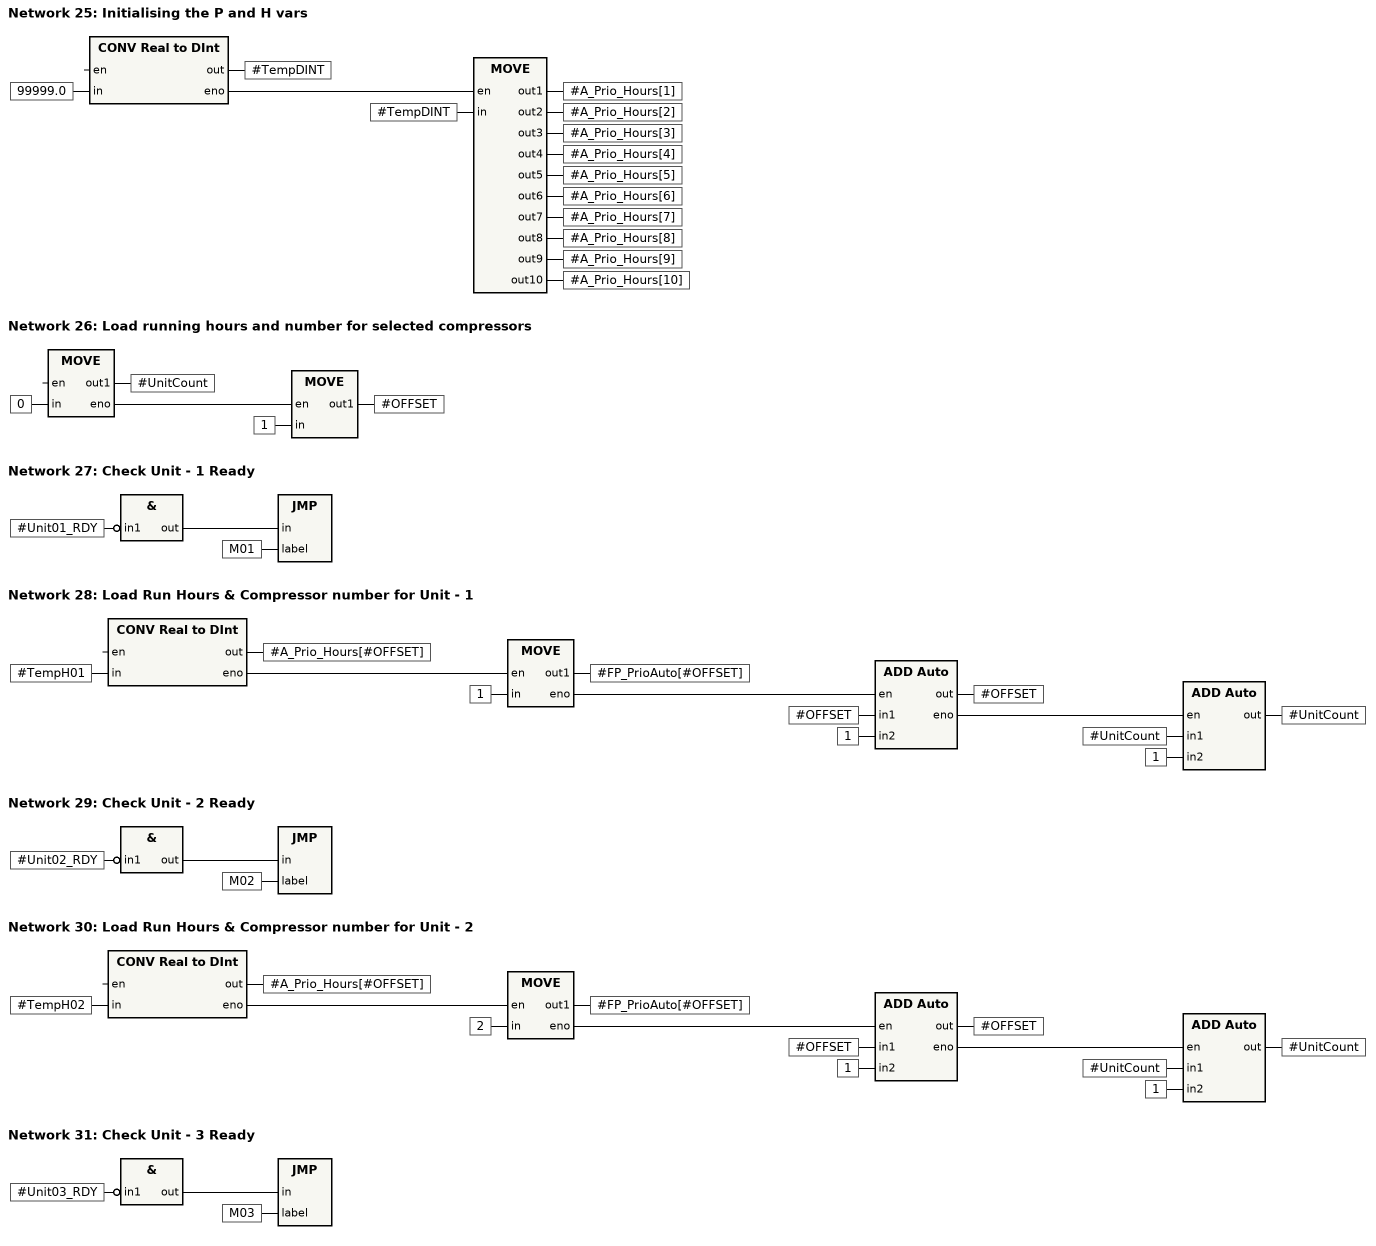
   #TempDINT := REAL_TO_DINT(99999.0);
   #A_Prio_Hours[1] := #TempDINT;
   #A_Prio_Hours[2] := #TempDINT;
   #A_Prio_Hours[3] := #TempDINT;
   #A_Prio_Hours[4] := #TempDINT;
   #A_Prio_Hours[5] := #TempDINT;
   #A_Prio_Hours[6] := #TempDINT;
   #A_Prio_Hours[7] := #TempDINT;
   #A_Prio_Hours[8] := #TempDINT;
   #A_Prio_Hours[9] := #TempDINT;
   #A_Prio_Hours[10] := #TempDINT;
END_REGION

REGION Network 26: Load running hours and number for selected compressors
   // Initialise Unit Count and Offset
   #UnitCount := 0;
   #OFFSET := 1;
END_REGION

REGION Network 27: Check Unit - 1 Ready
   IF NOT #Unit01_RDY THEN GOTO M01; END_IF;
END_REGION

REGION Network 28: Load Run Hours & Compressor number for Unit - 1
   #A_Prio_Hours[#OFFSET] := REAL_TO_DINT(#TempH01);
   #FP_PrioAuto[#OFFSET] := 1;
   #OFFSET := #OFFSET + 1;
   #UnitCount := #UnitCount + 1;
END_REGION

REGION Network 29: Check Unit - 2 Ready
   M01:
   IF NOT #Unit02_RDY THEN GOTO M02; END_IF;
END_REGION

REGION Network 30: Load Run Hours & Compressor number for Unit - 2
   #A_Prio_Hours[#OFFSET] := REAL_TO_DINT(#TempH02);
   #FP_PrioAuto[#OFFSET] := 2;
   #OFFSET := #OFFSET + 1;
   #UnitCount := #UnitCount + 1;
END_REGION

REGION Network 31: Check Unit - 3 Ready
   M02:
   IF NOT #Unit03_RDY THEN GOTO M03; END_IF;
END_REGION

REGION Network 32: Load Run Hours & Compressor number for Unit - 3
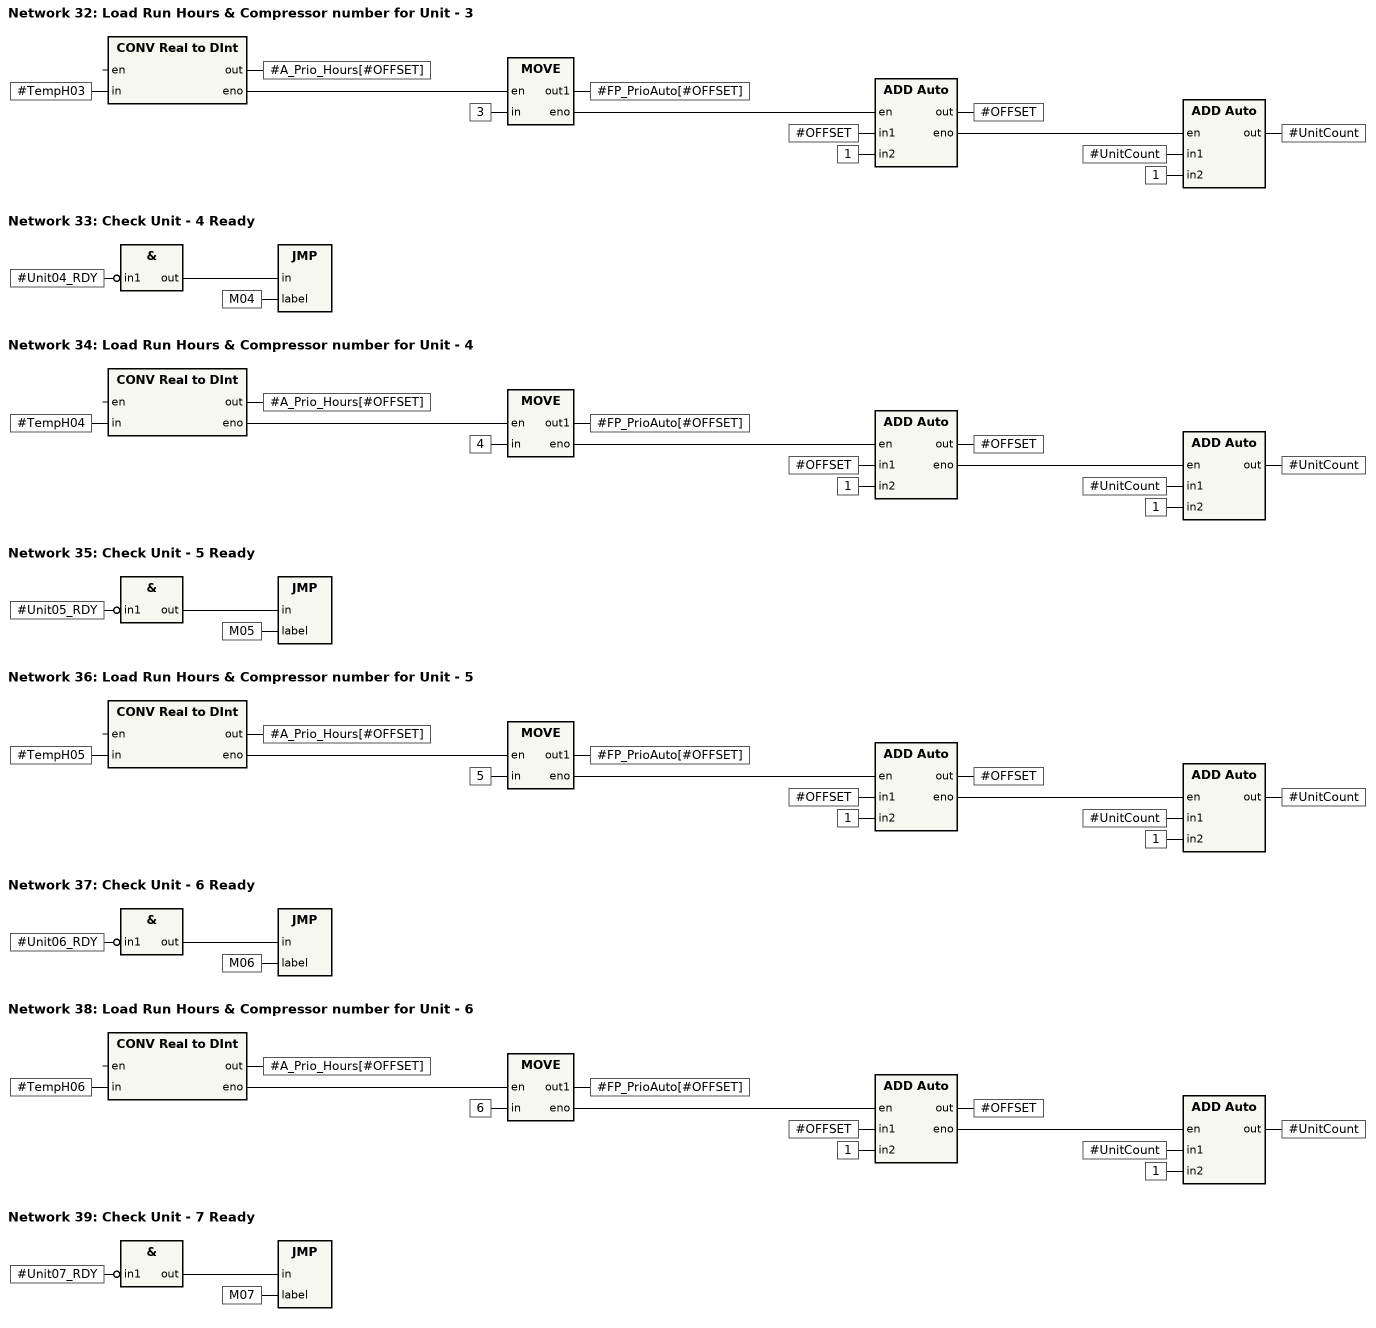
   #A_Prio_Hours[#OFFSET] := REAL_TO_DINT(#TempH03);
   #FP_PrioAuto[#OFFSET] := 3;
   #OFFSET := #OFFSET + 1;
   #UnitCount := #UnitCount + 1;
END_REGION

REGION Network 33: Check Unit - 4 Ready
   M03:
   IF NOT #Unit04_RDY THEN GOTO M04; END_IF;
END_REGION

REGION Network 34: Load Run Hours & Compressor number for Unit - 4
   #A_Prio_Hours[#OFFSET] := REAL_TO_DINT(#TempH04);
   #FP_PrioAuto[#OFFSET] := 4;
   #OFFSET := #OFFSET + 1;
   #UnitCount := #UnitCount + 1;
END_REGION

REGION Network 35: Check Unit - 5 Ready
   M04:
   IF NOT #Unit05_RDY THEN GOTO M05; END_IF;
END_REGION

REGION Network 36: Load Run Hours & Compressor number for Unit - 5
   #A_Prio_Hours[#OFFSET] := REAL_TO_DINT(#TempH05);
   #FP_PrioAuto[#OFFSET] := 5;
   #OFFSET := #OFFSET + 1;
   #UnitCount := #UnitCount + 1;
END_REGION

REGION Network 37: Check Unit - 6 Ready
   M05:
   IF NOT #Unit06_RDY THEN GOTO M06; END_IF;
END_REGION

REGION Network 38: Load Run Hours & Compressor number for Unit - 6
   #A_Prio_Hours[#OFFSET] := REAL_TO_DINT(#TempH06);
   #FP_PrioAuto[#OFFSET] := 6;
   #OFFSET := #OFFSET + 1;
   #UnitCount := #UnitCount + 1;
END_REGION

REGION Network 39: Check Unit - 7 Ready
   M06:
   IF NOT #Unit07_RDY THEN GOTO M07; END_IF;
END_REGION

REGION Network 40: Load Run Hours & Compressor number for Unit - 7
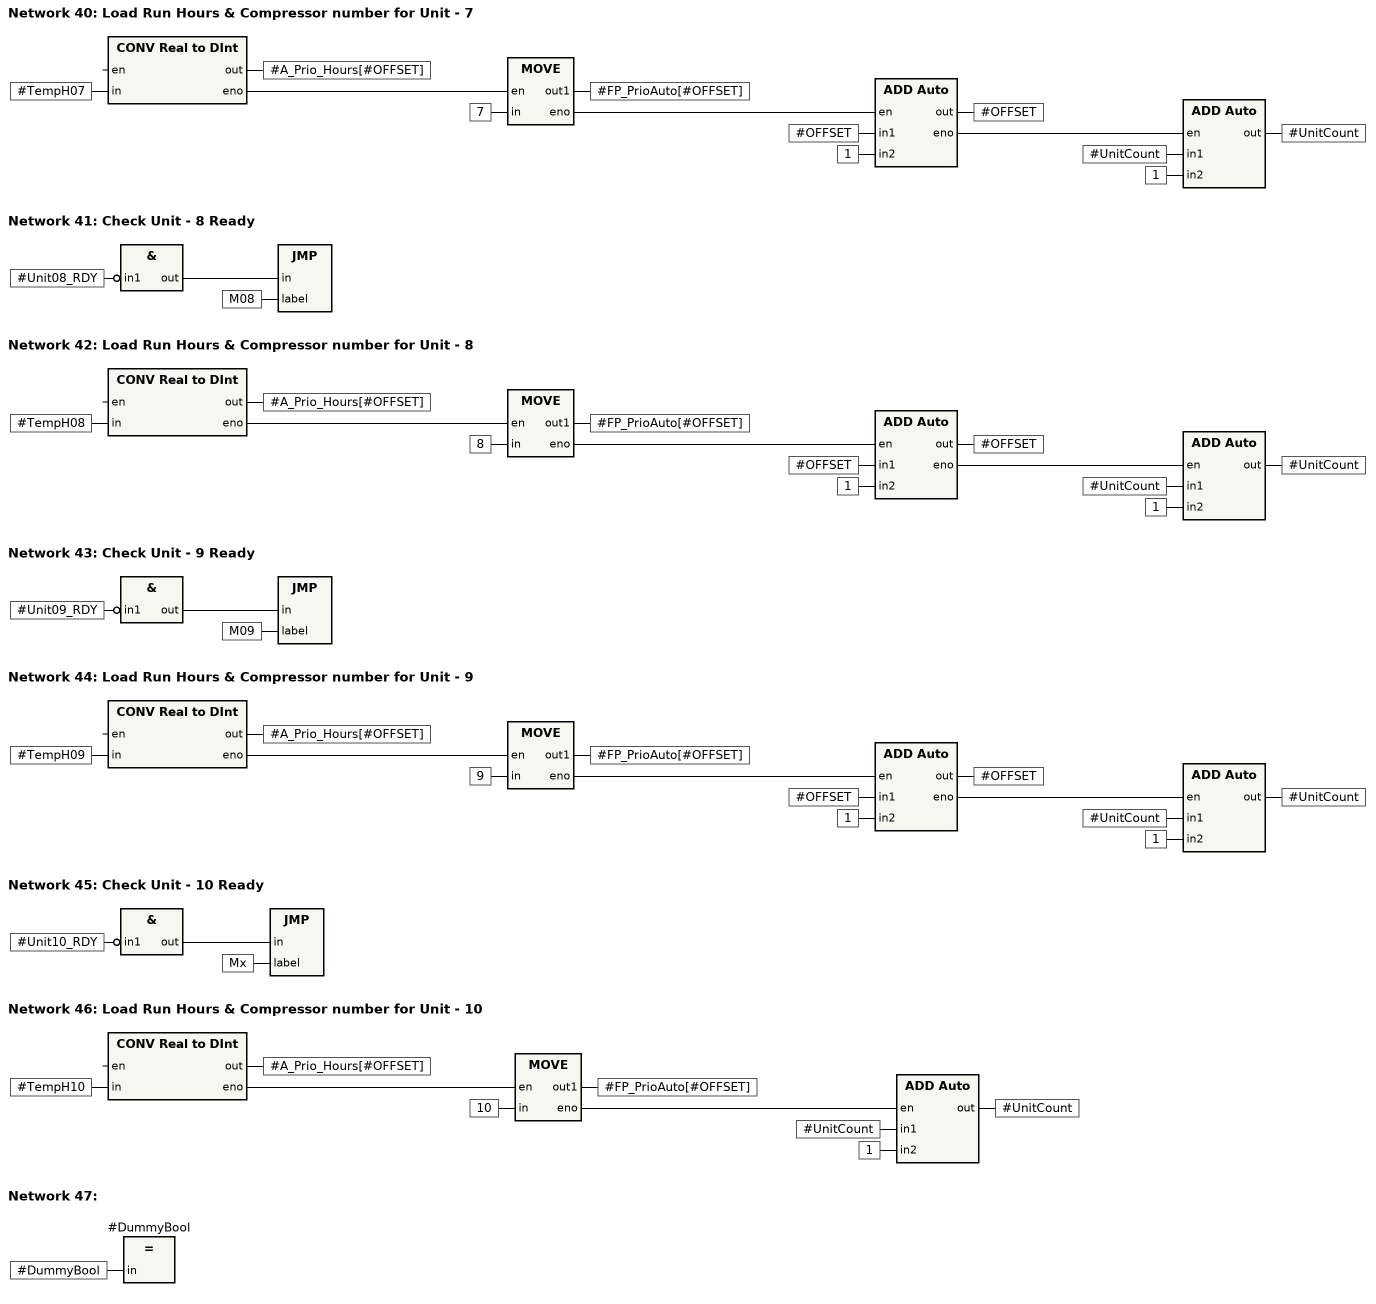
   #A_Prio_Hours[#OFFSET] := REAL_TO_DINT(#TempH07);
   #FP_PrioAuto[#OFFSET] := 7;
   #OFFSET := #OFFSET + 1;
   #UnitCount := #UnitCount + 1;
END_REGION

REGION Network 41: Check Unit - 8 Ready
   M07:
   IF NOT #Unit08_RDY THEN GOTO M08; END_IF;
END_REGION

REGION Network 42: Load Run Hours & Compressor number for Unit - 8
   #A_Prio_Hours[#OFFSET] := REAL_TO_DINT(#TempH08);
   #FP_PrioAuto[#OFFSET] := 8;
   #OFFSET := #OFFSET + 1;
   #UnitCount := #UnitCount + 1;
END_REGION

REGION Network 43: Check Unit - 9 Ready
   M08:
   IF NOT #Unit09_RDY THEN GOTO M09; END_IF;
END_REGION

REGION Network 44: Load Run Hours & Compressor number for Unit - 9
   #A_Prio_Hours[#OFFSET] := REAL_TO_DINT(#TempH09);
   #FP_PrioAuto[#OFFSET] := 9;
   #OFFSET := #OFFSET + 1;
   #UnitCount := #UnitCount + 1;
END_REGION

REGION Network 45: Check Unit - 10 Ready
   M09:
   IF NOT #Unit10_RDY THEN GOTO Mx; END_IF;
END_REGION

REGION Network 46: Load Run Hours & Compressor number for Unit - 10
   #A_Prio_Hours[#OFFSET] := REAL_TO_DINT(#TempH10);
   #FP_PrioAuto[#OFFSET] := 10;
   #UnitCount := #UnitCount + 1;
END_REGION

REGION Network 47
   Mx:
   #DummyBool := #DummyBool;
END_REGION

REGION Network 48: Bubbel Sort
   // The sort look at the current value compares this with the next, if the next 
   // value is less than the current they change places. After one full run thru 
   // the values without any changes the array is sorted.
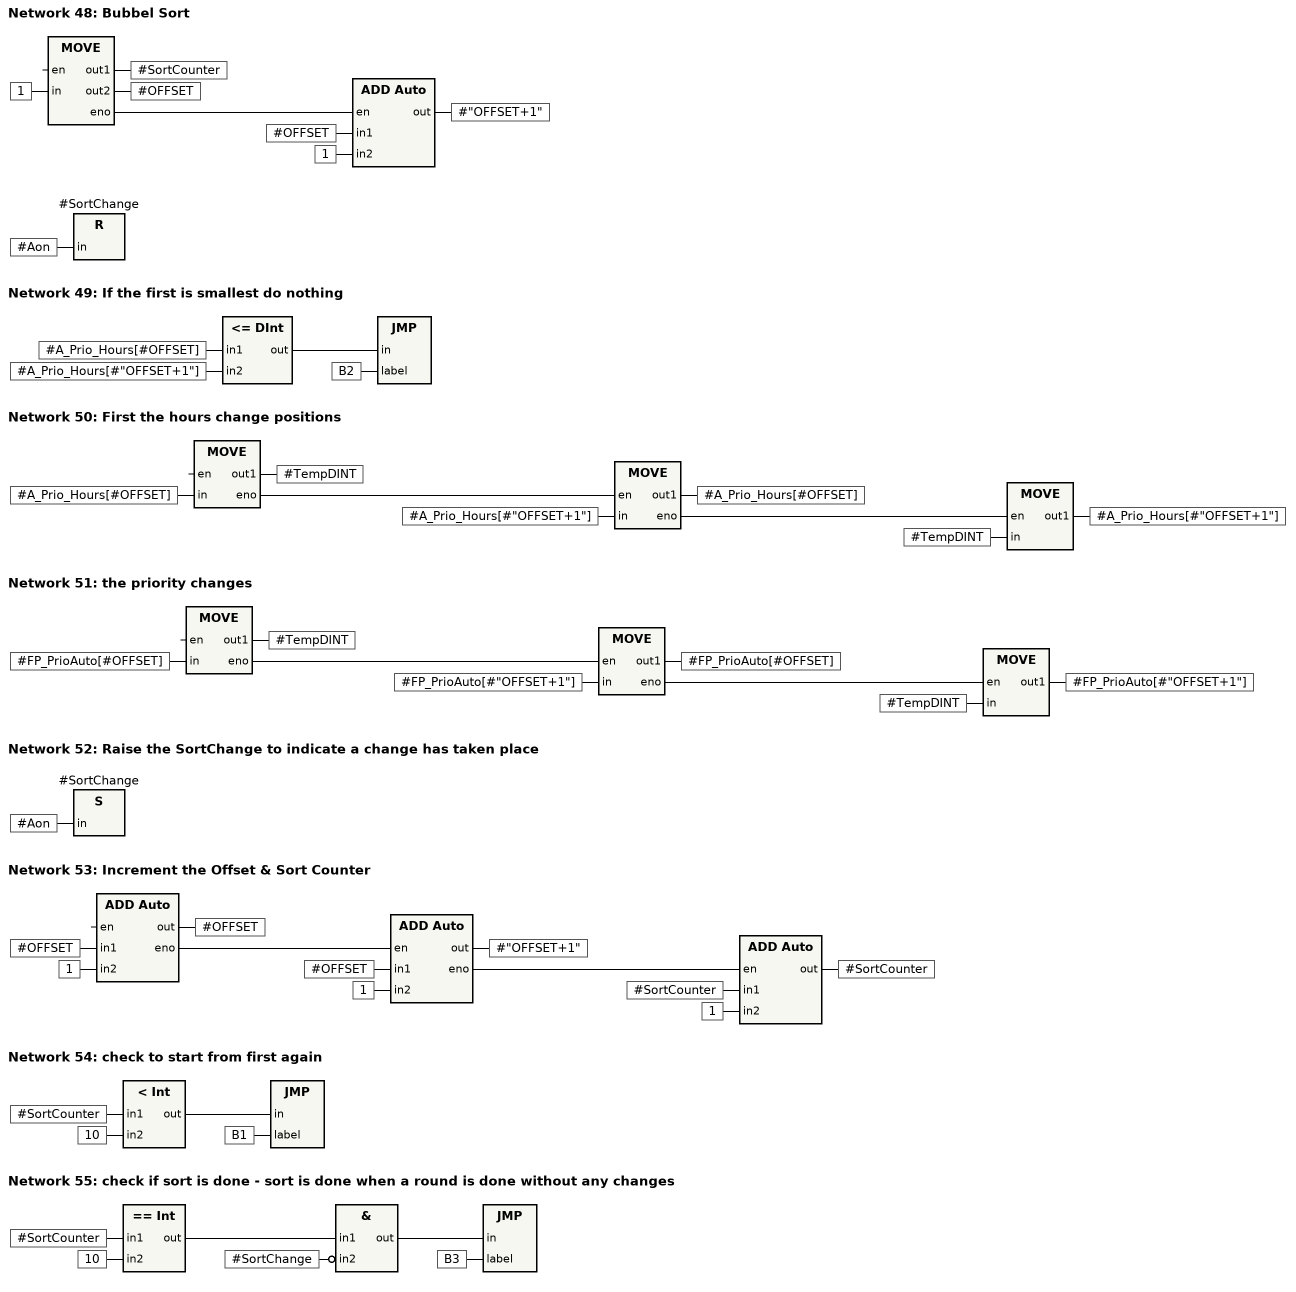
   #SortCounter := 1;
   #OFFSET := 1;
   #"OFFSET+1" := #OFFSET + 1;
   IF #Aon THEN #SortChange := FALSE; END_IF;
END_REGION

REGION Network 49: If the first is smallest do nothing
   B1:
   IF #A_Prio_Hours[#OFFSET] <= #A_Prio_Hours[#"OFFSET+1"] THEN GOTO B2; END_IF;
END_REGION

REGION Network 50: First the hours change positions
   #TempDINT := #A_Prio_Hours[#OFFSET];
   #A_Prio_Hours[#OFFSET] := #A_Prio_Hours[#"OFFSET+1"];
   #A_Prio_Hours[#"OFFSET+1"] := #TempDINT;
END_REGION

REGION Network 51: the priority changes
   #TempDINT := #FP_PrioAuto[#OFFSET];
   #FP_PrioAuto[#OFFSET] := #FP_PrioAuto[#"OFFSET+1"];
   #FP_PrioAuto[#"OFFSET+1"] := #TempDINT;
END_REGION

REGION Network 52: Raise the SortChange to indicate a change has taken place
   IF #Aon THEN #SortChange := TRUE; END_IF;
END_REGION

REGION Network 53: Increment the Offset & Sort Counter
   B2:
   #OFFSET := #OFFSET + 1;
   #"OFFSET+1" := #OFFSET + 1;
   #SortCounter := #SortCounter + 1;
END_REGION

REGION Network 54: check to start from first again
   IF #SortCounter < 10 THEN GOTO B1; END_IF;
END_REGION

REGION Network 55: check if sort is done - sort is done when a round is done without any changes
   IF (#SortCounter = 10) AND NOT #SortChange THEN GOTO B3; END_IF;
END_REGION

REGION Network 56: reset SortChange for new check
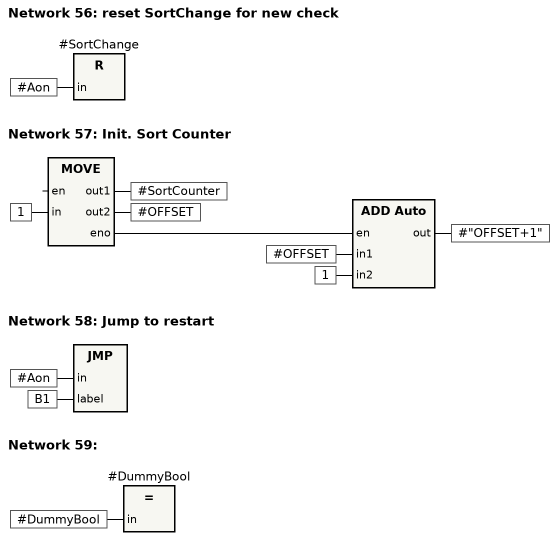
   IF #Aon THEN #SortChange := FALSE; END_IF;
END_REGION

REGION Network 57: Init. Sort Counter
   #SortCounter := 1;
   #OFFSET := 1;
   #"OFFSET+1" := #OFFSET + 1;
END_REGION

REGION Network 58: Jump to restart
   IF #Aon THEN GOTO B1; END_IF;
END_REGION

REGION Network 59
   B3:
   #DummyBool := #DummyBool;
END_REGION

REGION Network 60: 3) Sorting of manual priority
   // Create temp vars.
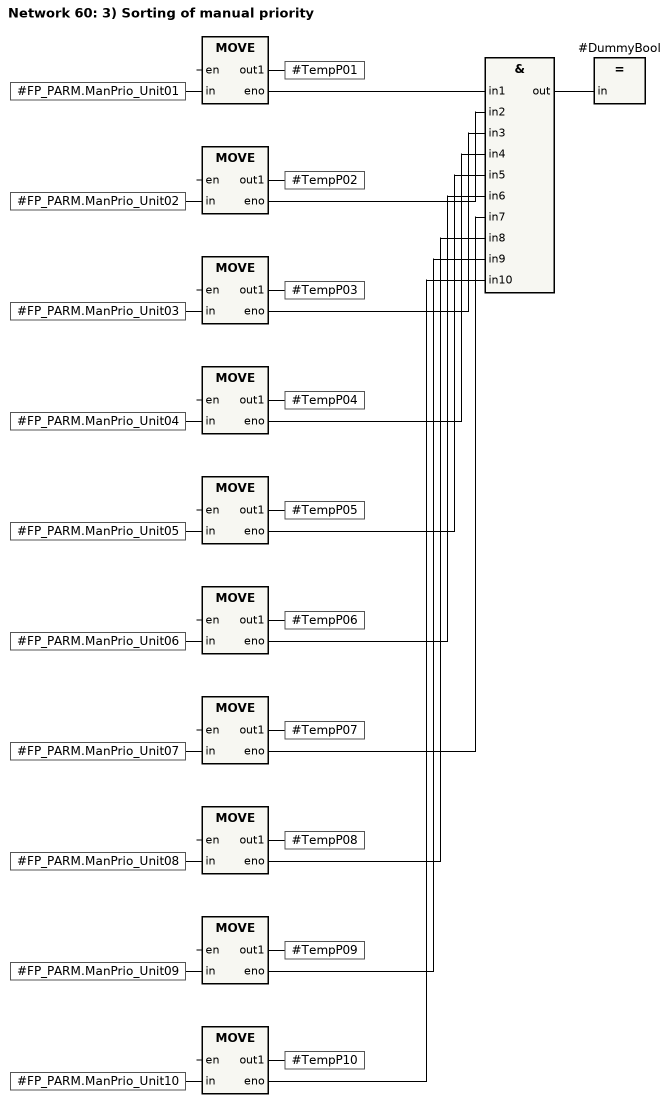
   #TempP01 := #FP_PARM.ManPrio_Unit01;
   #TempP02 := #FP_PARM.ManPrio_Unit02;
   #TempP03 := #FP_PARM.ManPrio_Unit03;
   #TempP04 := #FP_PARM.ManPrio_Unit04;
   #TempP05 := #FP_PARM.ManPrio_Unit05;
   #TempP06 := #FP_PARM.ManPrio_Unit06;
   #TempP07 := #FP_PARM.ManPrio_Unit07;
   #TempP08 := #FP_PARM.ManPrio_Unit08;
   #TempP09 := #FP_PARM.ManPrio_Unit09;
   #TempP10 := #FP_PARM.ManPrio_Unit10;
   #DummyBool := TRUE;
END_REGION

REGION Network 61: Initialising the MPN and MP vars
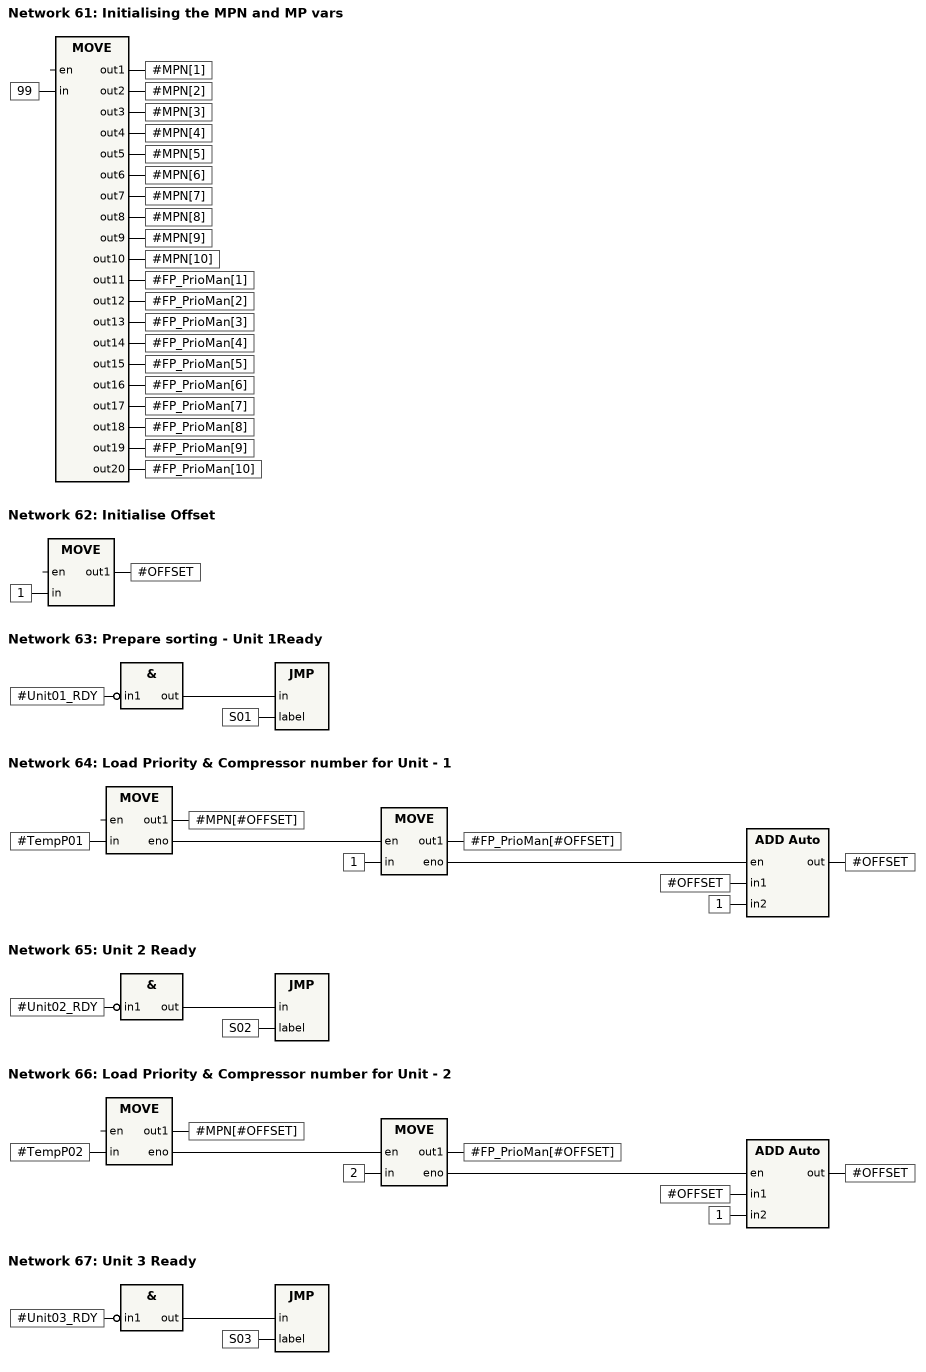
   #MPN[1] := 99;
   #MPN[2] := 99;
   #MPN[3] := 99;
   #MPN[4] := 99;
   #MPN[5] := 99;
   #MPN[6] := 99;
   #MPN[7] := 99;
   #MPN[8] := 99;
   #MPN[9] := 99;
   #MPN[10] := 99;
   #FP_PrioMan[1] := 99;
   #FP_PrioMan[2] := 99;
   #FP_PrioMan[3] := 99;
   #FP_PrioMan[4] := 99;
   #FP_PrioMan[5] := 99;
   #FP_PrioMan[6] := 99;
   #FP_PrioMan[7] := 99;
   #FP_PrioMan[8] := 99;
   #FP_PrioMan[9] := 99;
   #FP_PrioMan[10] := 99;
END_REGION

REGION Network 62: Initialise Offset
   #OFFSET := 1;
END_REGION

REGION Network 63: Prepare sorting - Unit 1Ready
   // If compressor isn't selected jump over
   IF NOT #Unit01_RDY THEN GOTO S01; END_IF;
END_REGION

REGION Network 64: Load Priority & Compressor number for Unit - 1
   // Load Priority and compressor number into arrays for sorting
   #MPN[#OFFSET] := #TempP01;
   #FP_PrioMan[#OFFSET] := 1;
   #OFFSET := #OFFSET + 1;
END_REGION

REGION Network 65: Unit 2 Ready
   S01:
   IF NOT #Unit02_RDY THEN GOTO S02; END_IF;
END_REGION

REGION Network 66: Load Priority & Compressor number for Unit - 2
   #MPN[#OFFSET] := #TempP02;
   #FP_PrioMan[#OFFSET] := 2;
   #OFFSET := #OFFSET + 1;
END_REGION

REGION Network 67: Unit 3 Ready
   S02:
   IF NOT #Unit03_RDY THEN GOTO S03; END_IF;
END_REGION

REGION Network 68: Load Priority & Compressor number for Unit - 3
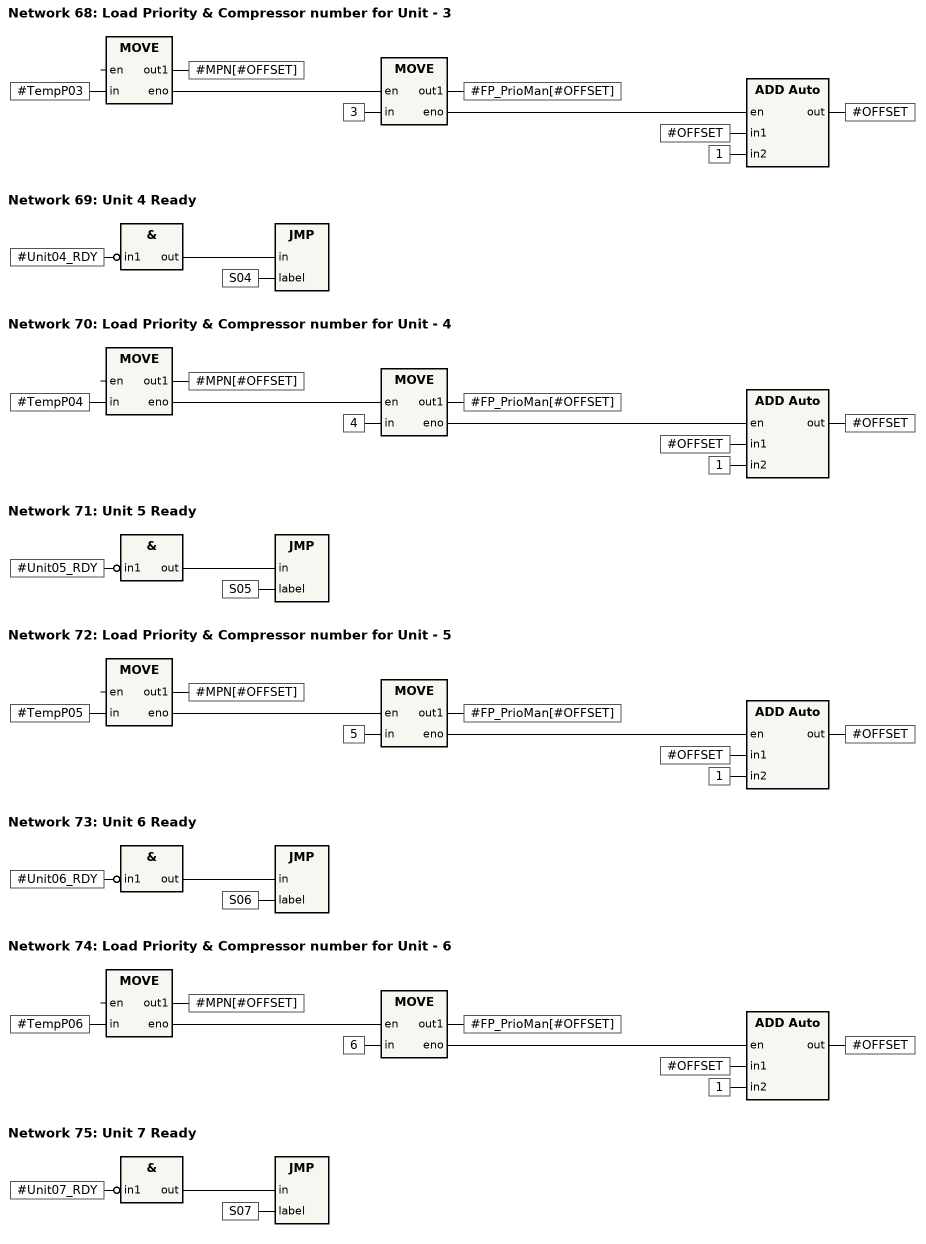
   #MPN[#OFFSET] := #TempP03;
   #FP_PrioMan[#OFFSET] := 3;
   #OFFSET := #OFFSET + 1;
END_REGION

REGION Network 69: Unit 4 Ready
   S03:
   IF NOT #Unit04_RDY THEN GOTO S04; END_IF;
END_REGION

REGION Network 70: Load Priority & Compressor number for Unit - 4
   #MPN[#OFFSET] := #TempP04;
   #FP_PrioMan[#OFFSET] := 4;
   #OFFSET := #OFFSET + 1;
END_REGION

REGION Network 71: Unit 5 Ready
   S04:
   IF NOT #Unit05_RDY THEN GOTO S05; END_IF;
END_REGION

REGION Network 72: Load Priority & Compressor number for Unit - 5
   #MPN[#OFFSET] := #TempP05;
   #FP_PrioMan[#OFFSET] := 5;
   #OFFSET := #OFFSET + 1;
END_REGION

REGION Network 73: Unit 6 Ready
   S05:
   IF NOT #Unit06_RDY THEN GOTO S06; END_IF;
END_REGION

REGION Network 74: Load Priority & Compressor number for Unit - 6
   #MPN[#OFFSET] := #TempP06;
   #FP_PrioMan[#OFFSET] := 6;
   #OFFSET := #OFFSET + 1;
END_REGION

REGION Network 75: Unit 7 Ready
   S06:
   IF NOT #Unit07_RDY THEN GOTO S07; END_IF;
END_REGION

REGION Network 76: Load Priority & Compressor number for Unit - 7
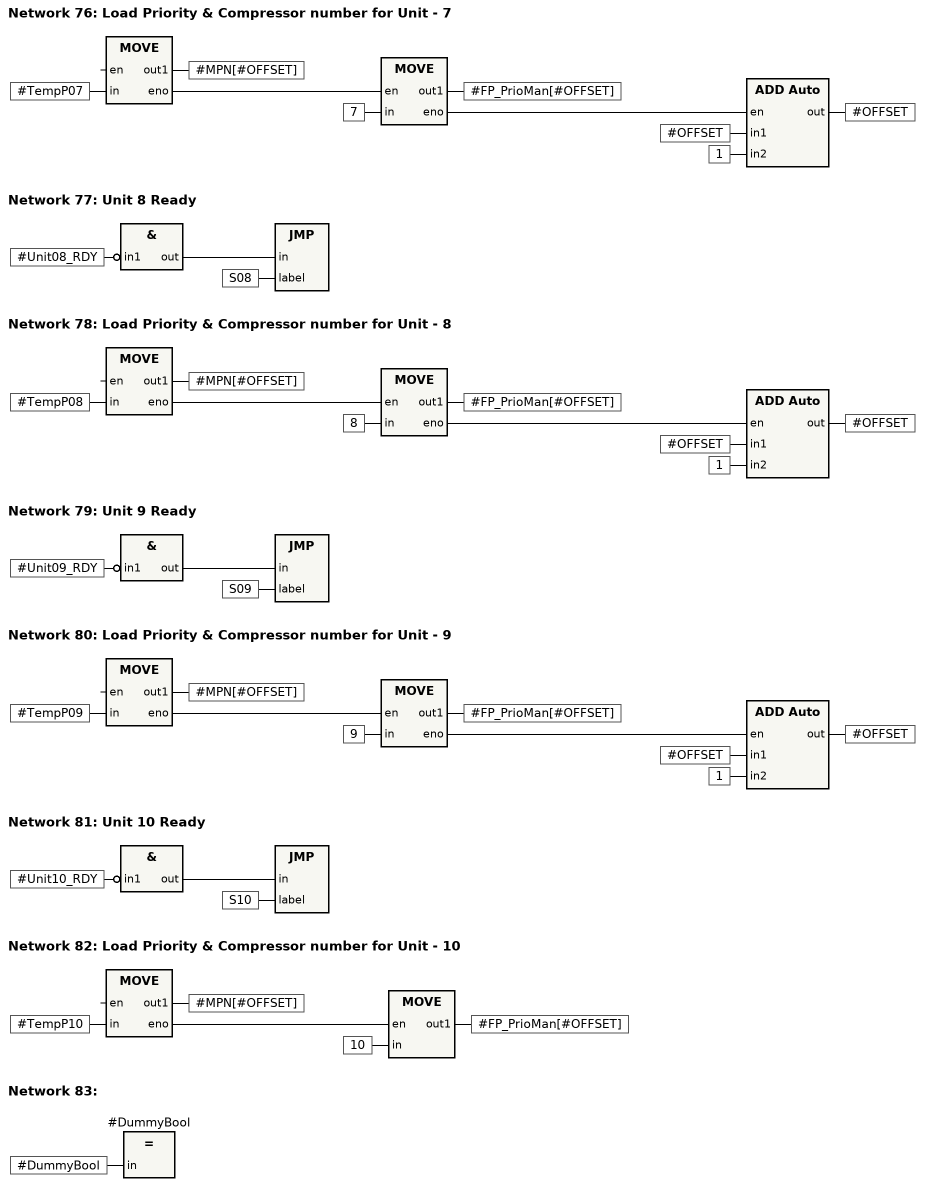
   #MPN[#OFFSET] := #TempP07;
   #FP_PrioMan[#OFFSET] := 7;
   #OFFSET := #OFFSET + 1;
END_REGION

REGION Network 77: Unit 8 Ready
   S07:
   IF NOT #Unit08_RDY THEN GOTO S08; END_IF;
END_REGION

REGION Network 78: Load Priority & Compressor number for Unit - 8
   #MPN[#OFFSET] := #TempP08;
   #FP_PrioMan[#OFFSET] := 8;
   #OFFSET := #OFFSET + 1;
END_REGION

REGION Network 79: Unit 9 Ready
   S08:
   IF NOT #Unit09_RDY THEN GOTO S09; END_IF;
END_REGION

REGION Network 80: Load Priority & Compressor number for Unit - 9
   #MPN[#OFFSET] := #TempP09;
   #FP_PrioMan[#OFFSET] := 9;
   #OFFSET := #OFFSET + 1;
END_REGION

REGION Network 81: Unit 10 Ready
   S09:
   IF NOT #Unit10_RDY THEN GOTO S10; END_IF;
END_REGION

REGION Network 82: Load Priority & Compressor number for Unit - 10
   #MPN[#OFFSET] := #TempP10;
   #FP_PrioMan[#OFFSET] := 10;
END_REGION

REGION Network 83
   S10:
   #DummyBool := #DummyBool;
END_REGION

REGION Network 84: Bubbel Sort manual priority
   // The sort look at the current value compares this with the next, if the next 
   // value is less than the current they change places. After one full run thru 
   // the values without any changes the array is sorted.
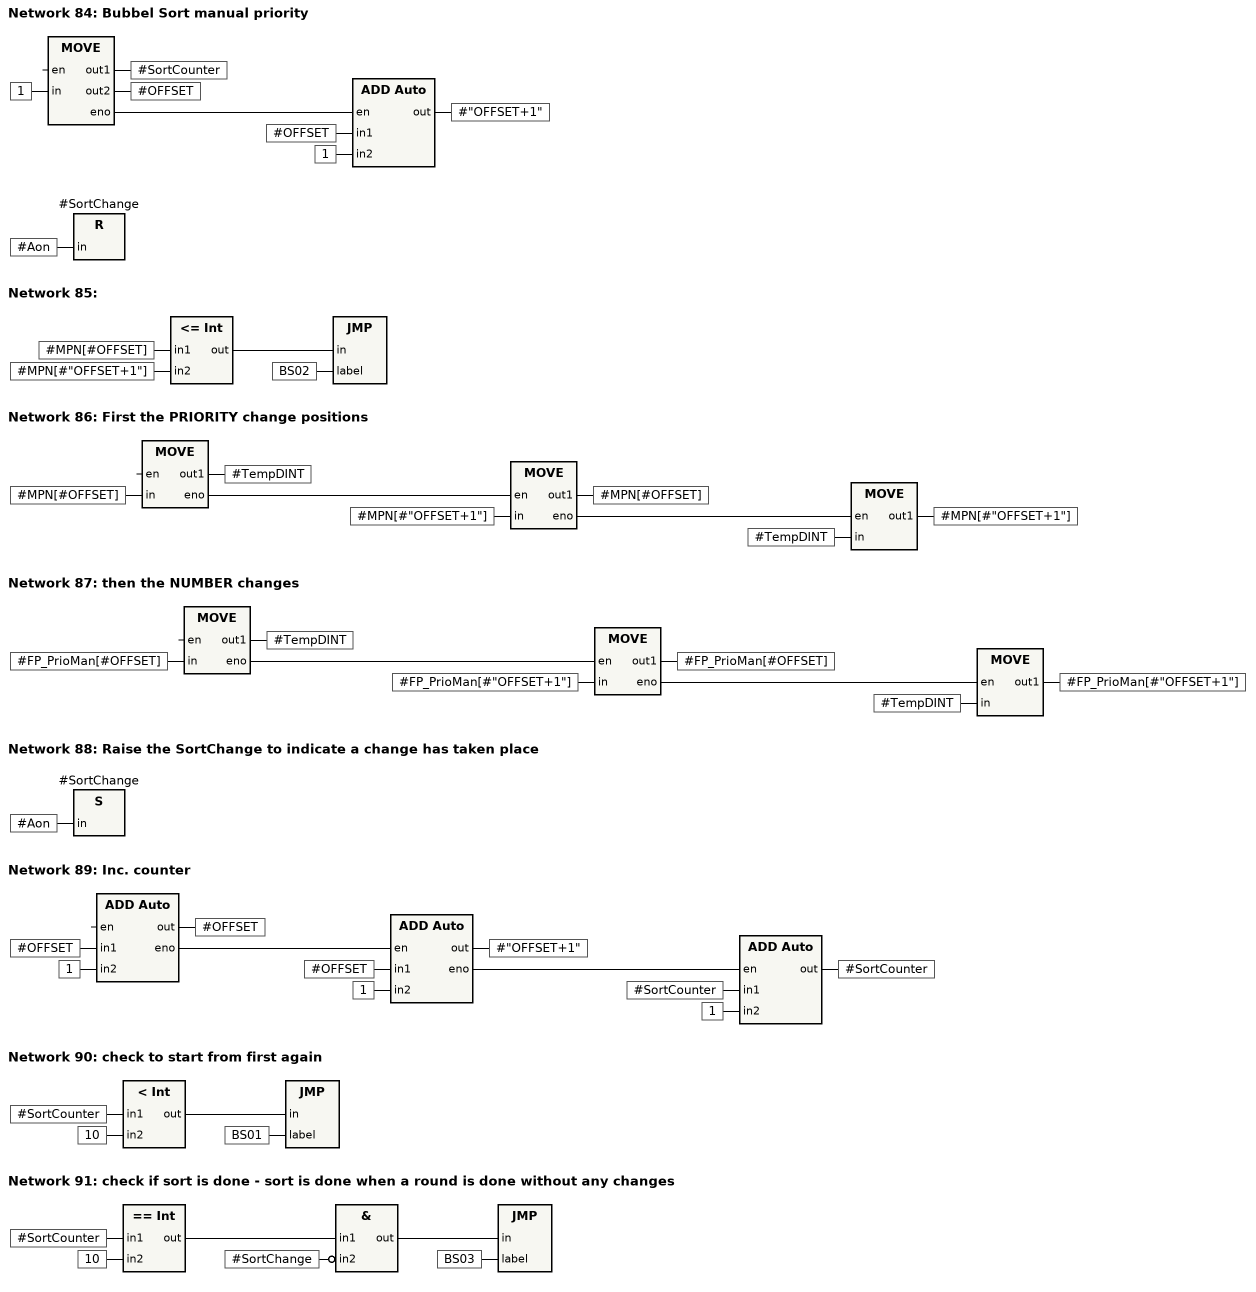
   #SortCounter := 1;
   #OFFSET := 1;
   #"OFFSET+1" := #OFFSET + 1;
   IF #Aon THEN #SortChange := FALSE; END_IF;
END_REGION

REGION Network 85
   // If the first is smallest do nothing
   BS01:
   IF #MPN[#OFFSET] <= #MPN[#"OFFSET+1"] THEN GOTO BS02; END_IF;
END_REGION

REGION Network 86: First the PRIORITY change positions
   #TempDINT := #MPN[#OFFSET];
   #MPN[#OFFSET] := #MPN[#"OFFSET+1"];
   #MPN[#"OFFSET+1"] := #TempDINT;
END_REGION

REGION Network 87: then the NUMBER changes
   #TempDINT := #FP_PrioMan[#OFFSET];
   #FP_PrioMan[#OFFSET] := #FP_PrioMan[#"OFFSET+1"];
   #FP_PrioMan[#"OFFSET+1"] := #TempDINT;
END_REGION

REGION Network 88: Raise the SortChange to indicate a change has taken place
   IF #Aon THEN #SortChange := TRUE; END_IF;
END_REGION

REGION Network 89: Inc. counter
   BS02:
   #OFFSET := #OFFSET + 1;
   #"OFFSET+1" := #OFFSET + 1;
   #SortCounter := #SortCounter + 1;
END_REGION

REGION Network 90: check to start from first again
   IF #SortCounter < 10 THEN GOTO BS01; END_IF;
END_REGION

REGION Network 91: check if sort is done - sort is done when a round is done without any changes
   IF (#SortCounter = 10) AND NOT #SortChange THEN GOTO BS03; END_IF;
END_REGION

REGION Network 92: reset SortChange for new check
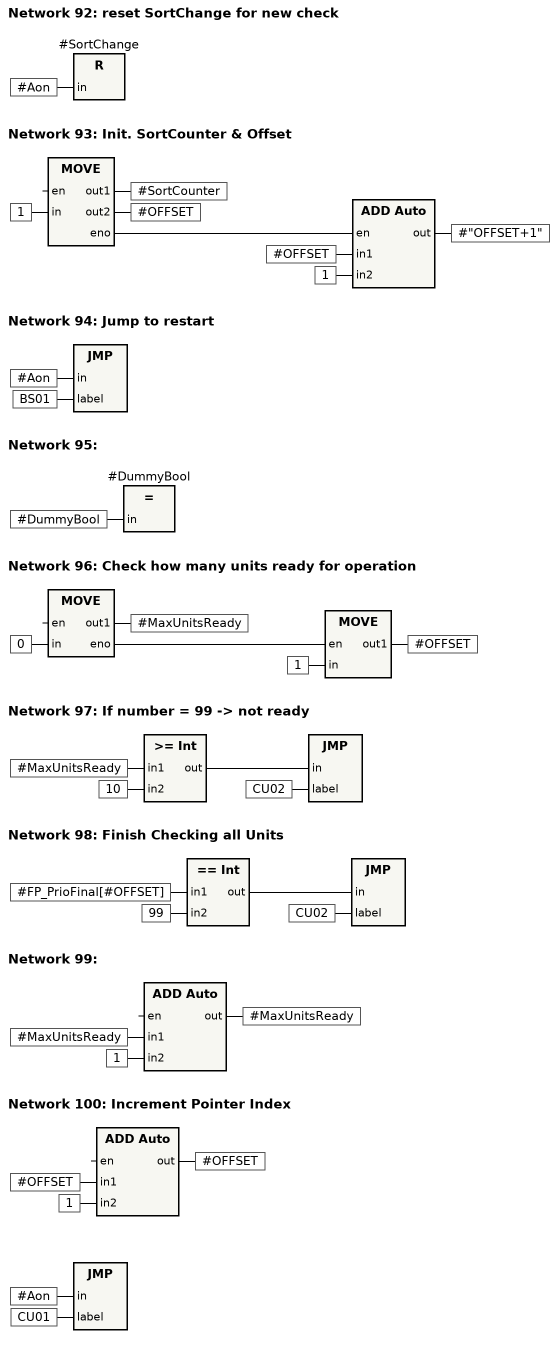
   IF #Aon THEN #SortChange := FALSE; END_IF;
END_REGION

REGION Network 93: Init. SortCounter & Offset
   #SortCounter := 1;
   #OFFSET := 1;
   #"OFFSET+1" := #OFFSET + 1;
END_REGION

REGION Network 94: Jump to restart
   IF #Aon THEN GOTO BS01; END_IF;
END_REGION

REGION Network 95
   BS03:
   #DummyBool := #DummyBool;
END_REGION

REGION Network 96: Check how many units ready for operation
   #MaxUnitsReady := 0;
   #OFFSET := 1;
END_REGION

REGION Network 97: If number = 99 -> not ready
   // Done, no more units ready
   // Build 003 - 11 Jul 2019 (EXTBOB) : Swapped this network with below network to avoid Area Length Error due to FP_PrioFinal wrong indexed
   CU01:
   IF #MaxUnitsReady >= 10 THEN GOTO CU02; END_IF;
END_REGION

REGION Network 98: Finish Checking all Units
   IF #FP_PrioFinal[#OFFSET] = 99 THEN GOTO CU02; END_IF;
END_REGION

REGION Network 99
   #MaxUnitsReady := #MaxUnitsReady + 1;
END_REGION

REGION Network 100: Increment Pointer Index
   #OFFSET := #OFFSET + 1;
   IF #Aon THEN GOTO CU01; END_IF;
END_REGION

REGION Network 101
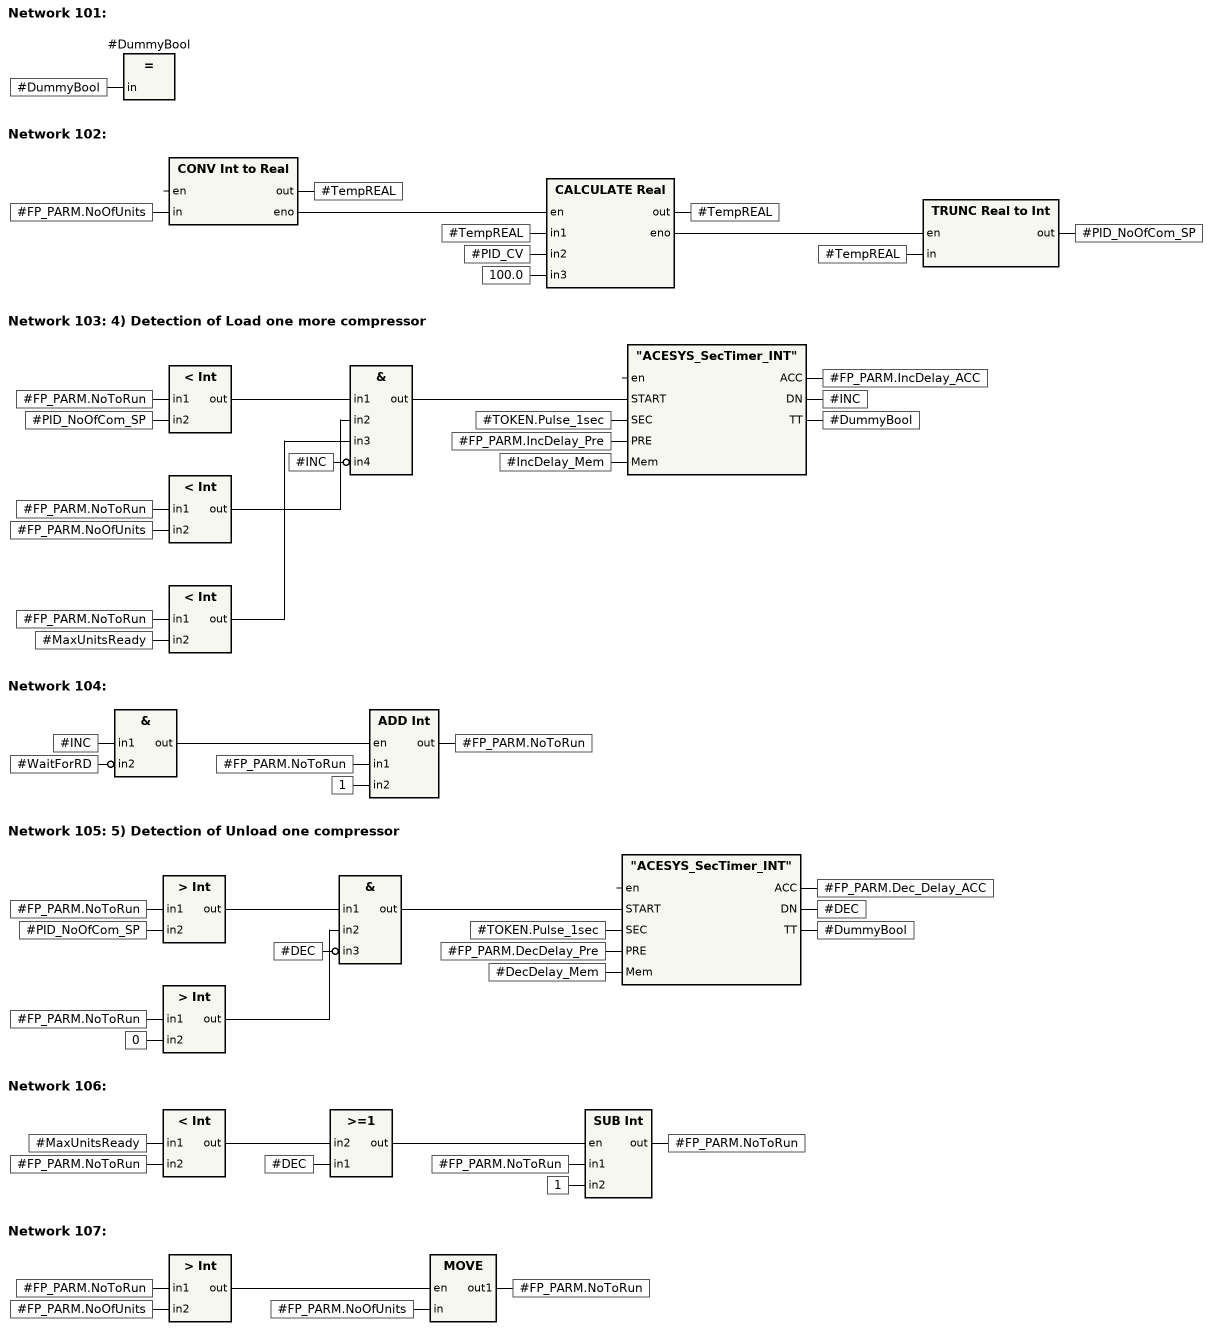
   CU02:
   #DummyBool := #DummyBool;
END_REGION

REGION Network 102
   #TempREAL := INT_TO_REAL(#FP_PARM.NoOfUnits);
   #TempREAL := (#TempREAL*#PID_CV)/100.0;
   #PID_NoOfCom_SP := TRUNC(#TempREAL);
END_REGION

REGION Network 103: 4) Detection of Load one more compressor
   // When the pressure has been below Low Limit for a longer time than set the next 
   // compressor starts.
   "ACESYS_SecTimer_INT"(START := (#FP_PARM.NoToRun < #PID_NoOfCom_SP) AND (#FP_PARM.NoToRun < #FP_PARM.NoOfUnits) AND (#FP_PARM.NoToRun < #MaxUnitsReady) AND NOT #INC,
                         SEC := #TOKEN.Pulse_1sec,
                         PRE := #FP_PARM.IncDelay_Pre,
                         Mem := #IncDelay_Mem,
                         ACC => #FP_PARM.IncDelay_ACC,
                         DN => #INC,
                         TT => #DummyBool);
END_REGION

REGION Network 104
   IF #INC AND NOT #WaitForRD THEN #FP_PARM.NoToRun := #FP_PARM.NoToRun + 1; END_IF;
END_REGION

REGION Network 105: 5) Detection of Unload one compressor
   // When the pressure has been above high Limit for a longer time than set a 
   // compressor stops.
   "ACESYS_SecTimer_INT"(START := (#FP_PARM.NoToRun > #PID_NoOfCom_SP) AND (#FP_PARM.NoToRun > 0) AND NOT #DEC,
                         SEC := #TOKEN.Pulse_1sec,
                         PRE := #FP_PARM.DecDelay_Pre,
                         Mem := #DecDelay_Mem,
                         ACC => #FP_PARM.Dec_Delay_ACC,
                         DN => #DEC,
                         TT => #DummyBool);
END_REGION

REGION Network 106
   IF (#MaxUnitsReady < #FP_PARM.NoToRun) OR #DEC THEN #FP_PARM.NoToRun := #FP_PARM.NoToRun - 1; END_IF;
END_REGION

REGION Network 107
   IF #FP_PARM.NoToRun > #FP_PARM.NoOfUnits THEN #FP_PARM.NoToRun := #FP_PARM.NoOfUnits; END_IF;
END_REGION

REGION Network 108: 6) Detection of priority change by timer in Auto
   // When in automatic priority mode the compressor pool is shifted according to 
   // running hours every x hours
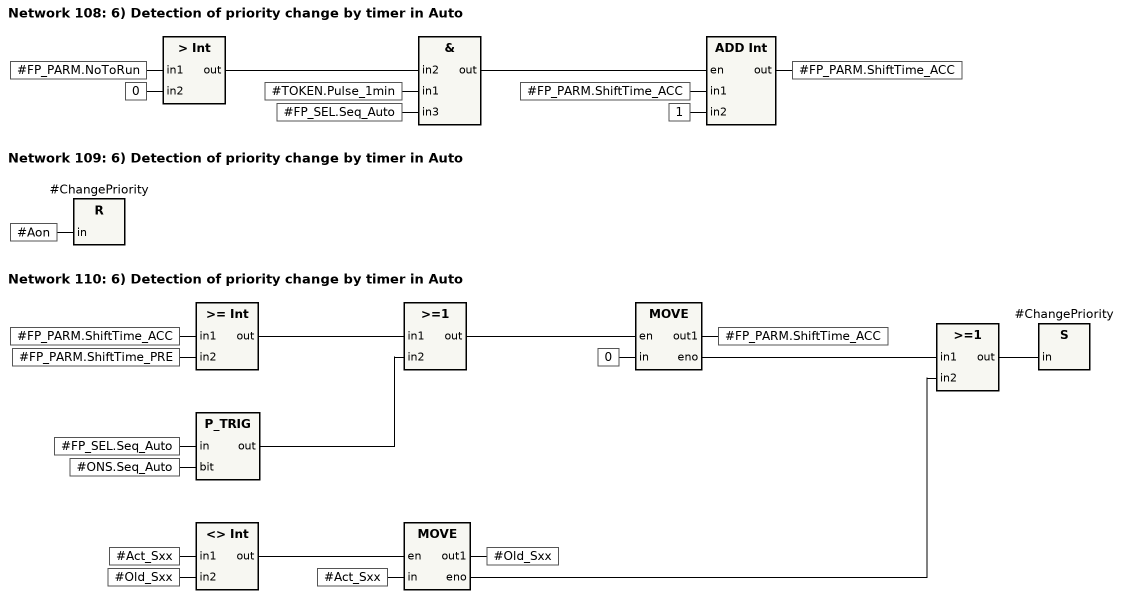
   IF (#FP_PARM.NoToRun > 0) AND #TOKEN.Pulse_1min AND #FP_SEL.Seq_Auto THEN
       #FP_PARM.ShiftTime_ACC := #FP_PARM.ShiftTime_ACC + 1;
   END_IF;
END_REGION

REGION Network 109: 6) Detection of priority change by timer in Auto
   IF #Aon THEN #ChangePriority := FALSE; END_IF;
END_REGION

REGION Network 110: 6) Detection of priority change by timer in Auto
   // ENO of a box is taken as its EN; it also drops when the box reports an error
   #_w1 := #FP_SEL.Seq_Auto AND NOT #ONS.Seq_Auto;   // rising edge
   #ONS.Seq_Auto := #FP_SEL.Seq_Auto;
   #_w2 := (#FP_PARM.ShiftTime_ACC >= #FP_PARM.ShiftTime_PRE) OR #_w1;
   IF #_w2 THEN #FP_PARM.ShiftTime_ACC := 0; END_IF;
   #_w3 := #Act_Sxx <> #Old_Sxx;
   IF #_w3 THEN #Old_Sxx := #Act_Sxx; END_IF;
   IF #_w2 OR #_w3 THEN #ChangePriority := TRUE; END_IF;
END_REGION

REGION Network 111: 7) Detect number of compresors running
   // In order to look up the compressor to load/unload the number of running 
   // compressors is detected. If the compressor is running and started by this 
   // routine then count
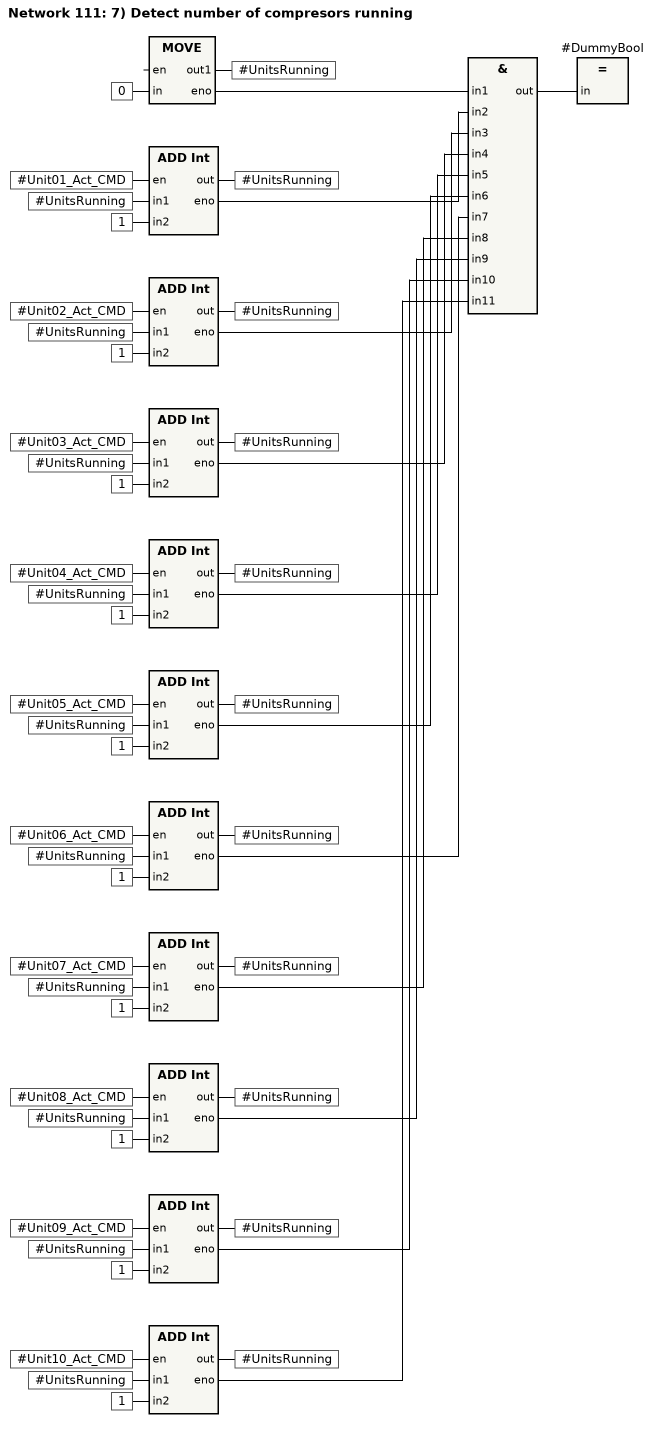
   // ENO of a box is taken as its EN; it also drops when the box reports an error
   #UnitsRunning := 0;
   IF #Unit01_Act_CMD THEN #UnitsRunning := #UnitsRunning + 1; END_IF;
   IF #Unit02_Act_CMD THEN #UnitsRunning := #UnitsRunning + 1; END_IF;
   IF #Unit03_Act_CMD THEN #UnitsRunning := #UnitsRunning + 1; END_IF;
   IF #Unit04_Act_CMD THEN #UnitsRunning := #UnitsRunning + 1; END_IF;
   IF #Unit05_Act_CMD THEN #UnitsRunning := #UnitsRunning + 1; END_IF;
   IF #Unit06_Act_CMD THEN #UnitsRunning := #UnitsRunning + 1; END_IF;
   IF #Unit07_Act_CMD THEN #UnitsRunning := #UnitsRunning + 1; END_IF;
   IF #Unit08_Act_CMD THEN #UnitsRunning := #UnitsRunning + 1; END_IF;
   IF #Unit09_Act_CMD THEN #UnitsRunning := #UnitsRunning + 1; END_IF;
   IF #Unit10_Act_CMD THEN #UnitsRunning := #UnitsRunning + 1; END_IF;
   #DummyBool := #Unit01_Act_CMD AND #Unit02_Act_CMD AND #Unit03_Act_CMD AND #Unit04_Act_CMD AND #Unit05_Act_CMD AND #Unit06_Act_CMD AND #Unit07_Act_CMD AND #Unit08_Act_CMD AND #Unit09_Act_CMD AND #Unit10_Act_CMD;
END_REGION

REGION Network 112: 8) Create final priority acording to selected mode (Manual)
   // If manual is selected then use the priority from ECS othervise use the one 
   // sorted out earlier in this program.
   // 
   // When using the manual the input must be sorted in the same way as the one based 
   // on automatic mode. i.e. the lowest priority in the buttom
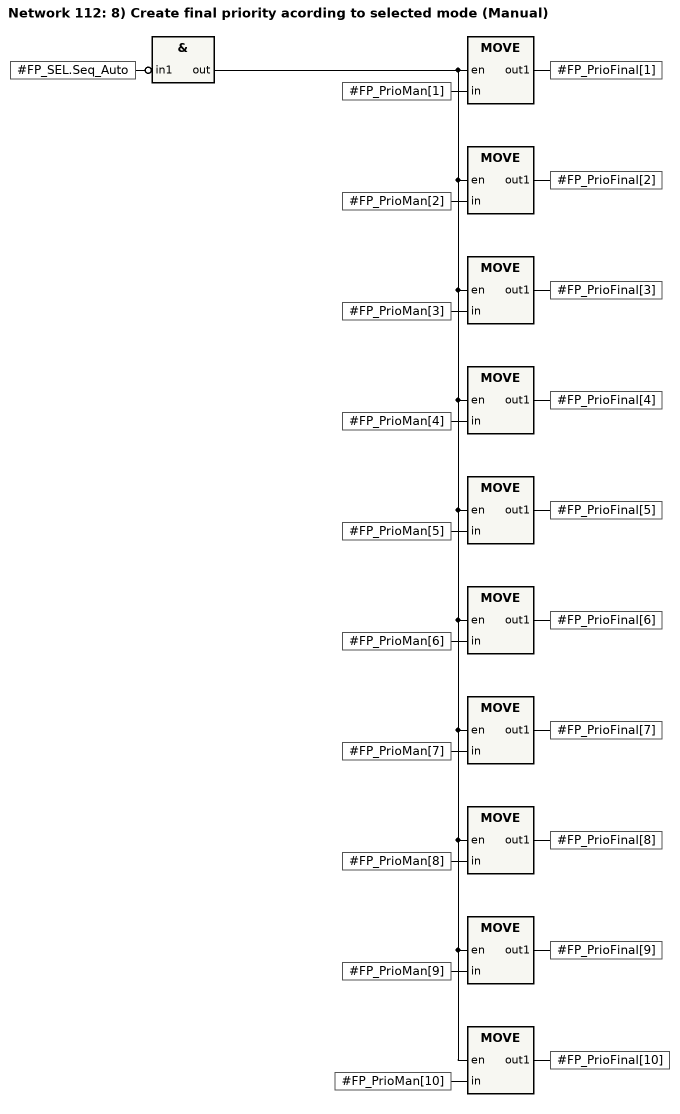
   IF NOT #FP_SEL.Seq_Auto THEN
       #FP_PrioFinal[1] := #FP_PrioMan[1];
       #FP_PrioFinal[2] := #FP_PrioMan[2];
       #FP_PrioFinal[3] := #FP_PrioMan[3];
       #FP_PrioFinal[4] := #FP_PrioMan[4];
       #FP_PrioFinal[5] := #FP_PrioMan[5];
       #FP_PrioFinal[6] := #FP_PrioMan[6];
       #FP_PrioFinal[7] := #FP_PrioMan[7];
       #FP_PrioFinal[8] := #FP_PrioMan[8];
       #FP_PrioFinal[9] := #FP_PrioMan[9];
       #FP_PrioFinal[10] := #FP_PrioMan[10];
   END_IF;
END_REGION

REGION Network 113: 8) Create final priority acording to selected mode (Auto)
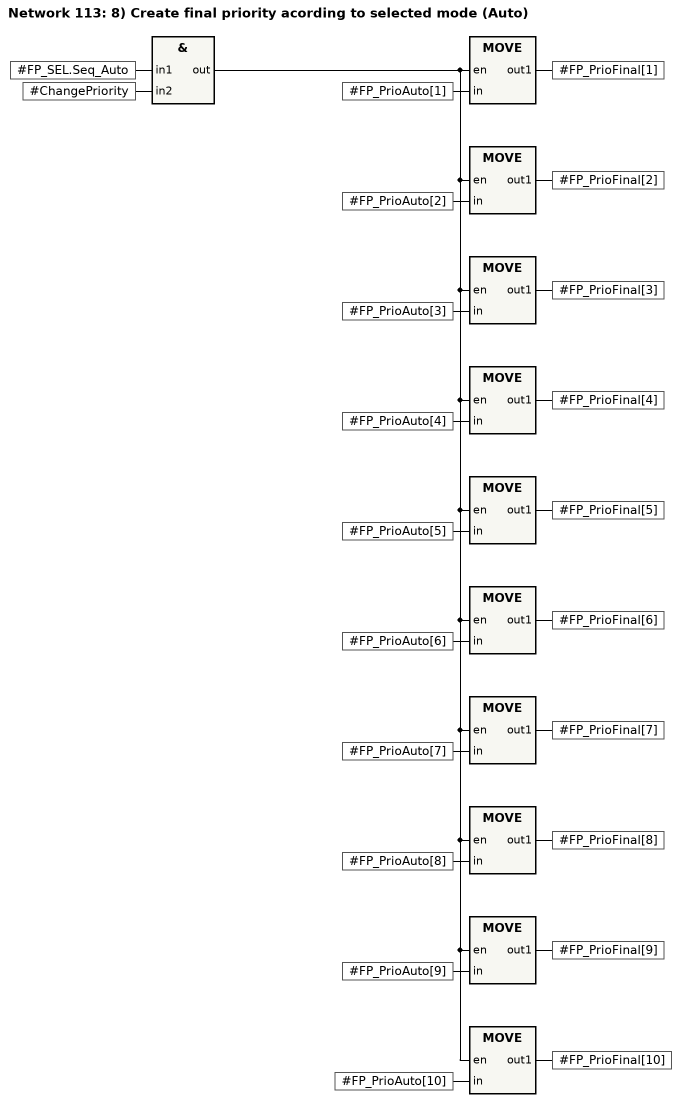
   IF #FP_SEL.Seq_Auto AND #ChangePriority THEN
       #FP_PrioFinal[1] := #FP_PrioAuto[1];
       #FP_PrioFinal[2] := #FP_PrioAuto[2];
       #FP_PrioFinal[3] := #FP_PrioAuto[3];
       #FP_PrioFinal[4] := #FP_PrioAuto[4];
       #FP_PrioFinal[5] := #FP_PrioAuto[5];
       #FP_PrioFinal[6] := #FP_PrioAuto[6];
       #FP_PrioFinal[7] := #FP_PrioAuto[7];
       #FP_PrioFinal[8] := #FP_PrioAuto[8];
       #FP_PrioFinal[9] := #FP_PrioAuto[9];
       #FP_PrioFinal[10] := #FP_PrioAuto[10];
   END_IF;
END_REGION

REGION Network 114: 9) Create ASTR command
   // In each scan the number of needed compressors are compared with the final 
   // priority in order to determine which compresors have to run
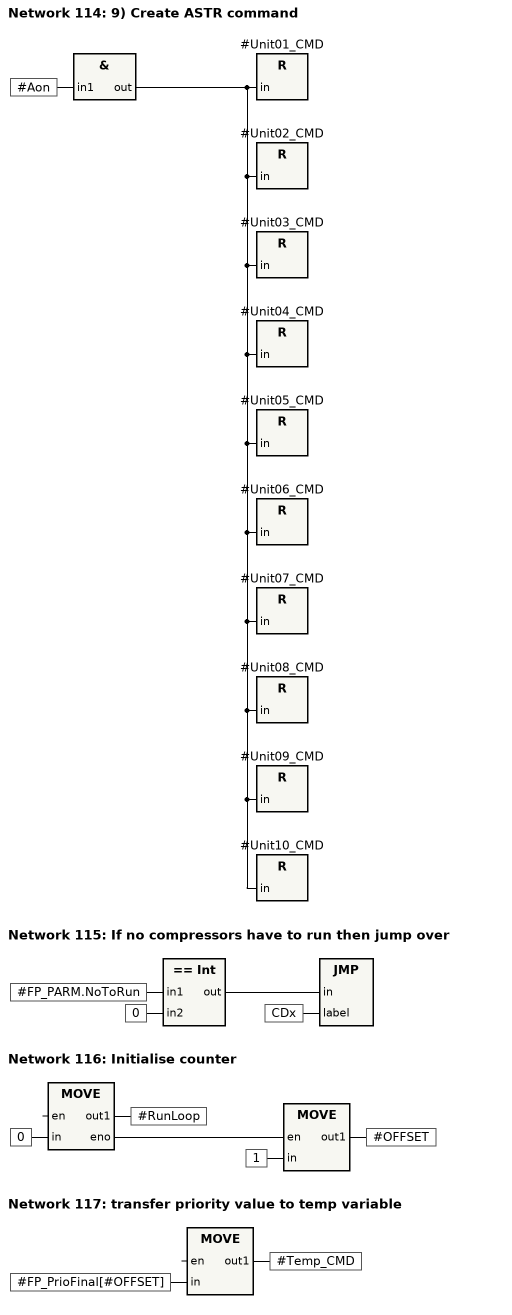
   IF #Aon THEN
       #Unit01_CMD := FALSE;
       #Unit02_CMD := FALSE;
       #Unit03_CMD := FALSE;
       #Unit04_CMD := FALSE;
       #Unit05_CMD := FALSE;
       #Unit06_CMD := FALSE;
       #Unit07_CMD := FALSE;
       #Unit08_CMD := FALSE;
       #Unit09_CMD := FALSE;
       #Unit10_CMD := FALSE;
   END_IF;
END_REGION

REGION Network 115: If no compressors have to run then jump over
   IF #FP_PARM.NoToRun = 0 THEN GOTO CDx; END_IF;
END_REGION

REGION Network 116: Initialise counter
   #RunLoop := 0;
   #OFFSET := 1;
END_REGION

REGION Network 117: transfer priority value to temp variable
   CD01:
   #Temp_CMD := #FP_PrioFinal[#OFFSET];
END_REGION

REGION Network 118: If the number in the final priority cell is different from the compressor number then jump over
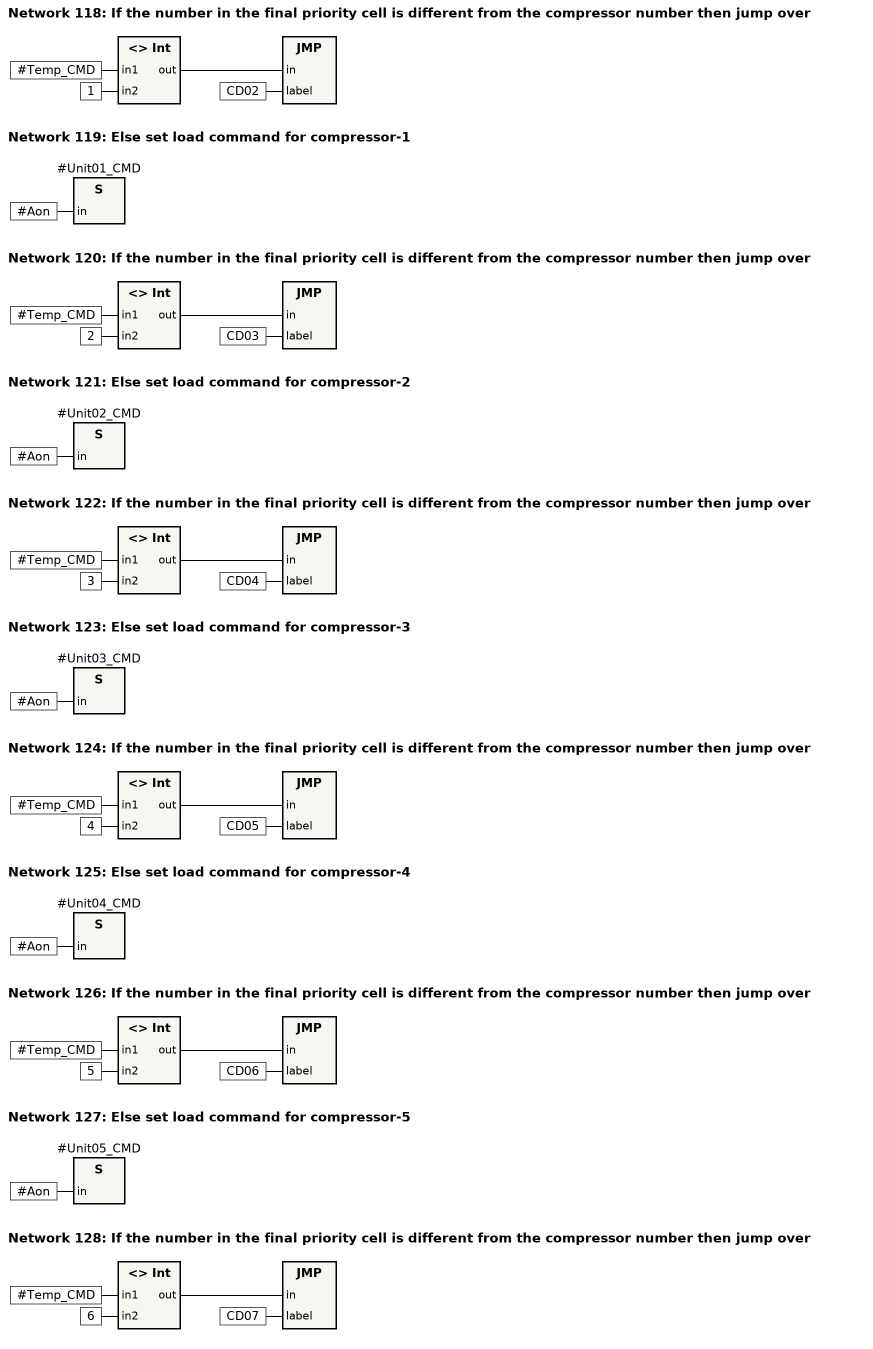
   IF #Temp_CMD <> 1 THEN GOTO CD02; END_IF;
END_REGION

REGION Network 119: Else set load command for compressor-1
   IF #Aon THEN #Unit01_CMD := TRUE; END_IF;
END_REGION

REGION Network 120: If the number in the final priority cell is different from the compressor number then jump over
   CD02:
   IF #Temp_CMD <> 2 THEN GOTO CD03; END_IF;
END_REGION

REGION Network 121: Else set load command for compressor-2
   IF #Aon THEN #Unit02_CMD := TRUE; END_IF;
END_REGION

REGION Network 122: If the number in the final priority cell is different from the compressor number then jump over
   CD03:
   IF #Temp_CMD <> 3 THEN GOTO CD04; END_IF;
END_REGION

REGION Network 123: Else set load command for compressor-3
   IF #Aon THEN #Unit03_CMD := TRUE; END_IF;
END_REGION

REGION Network 124: If the number in the final priority cell is different from the compressor number then jump over
   CD04:
   IF #Temp_CMD <> 4 THEN GOTO CD05; END_IF;
END_REGION

REGION Network 125: Else set load command for compressor-4
   IF #Aon THEN #Unit04_CMD := TRUE; END_IF;
END_REGION

REGION Network 126: If the number in the final priority cell is different from the compressor number then jump over
   CD05:
   IF #Temp_CMD <> 5 THEN GOTO CD06; END_IF;
END_REGION

REGION Network 127: Else set load command for compressor-5
   IF #Aon THEN #Unit05_CMD := TRUE; END_IF;
END_REGION

REGION Network 128: If the number in the final priority cell is different from the compressor number then jump over
   CD06:
   IF #Temp_CMD <> 6 THEN GOTO CD07; END_IF;
END_REGION

REGION Network 129: Else set load command for compressor-6
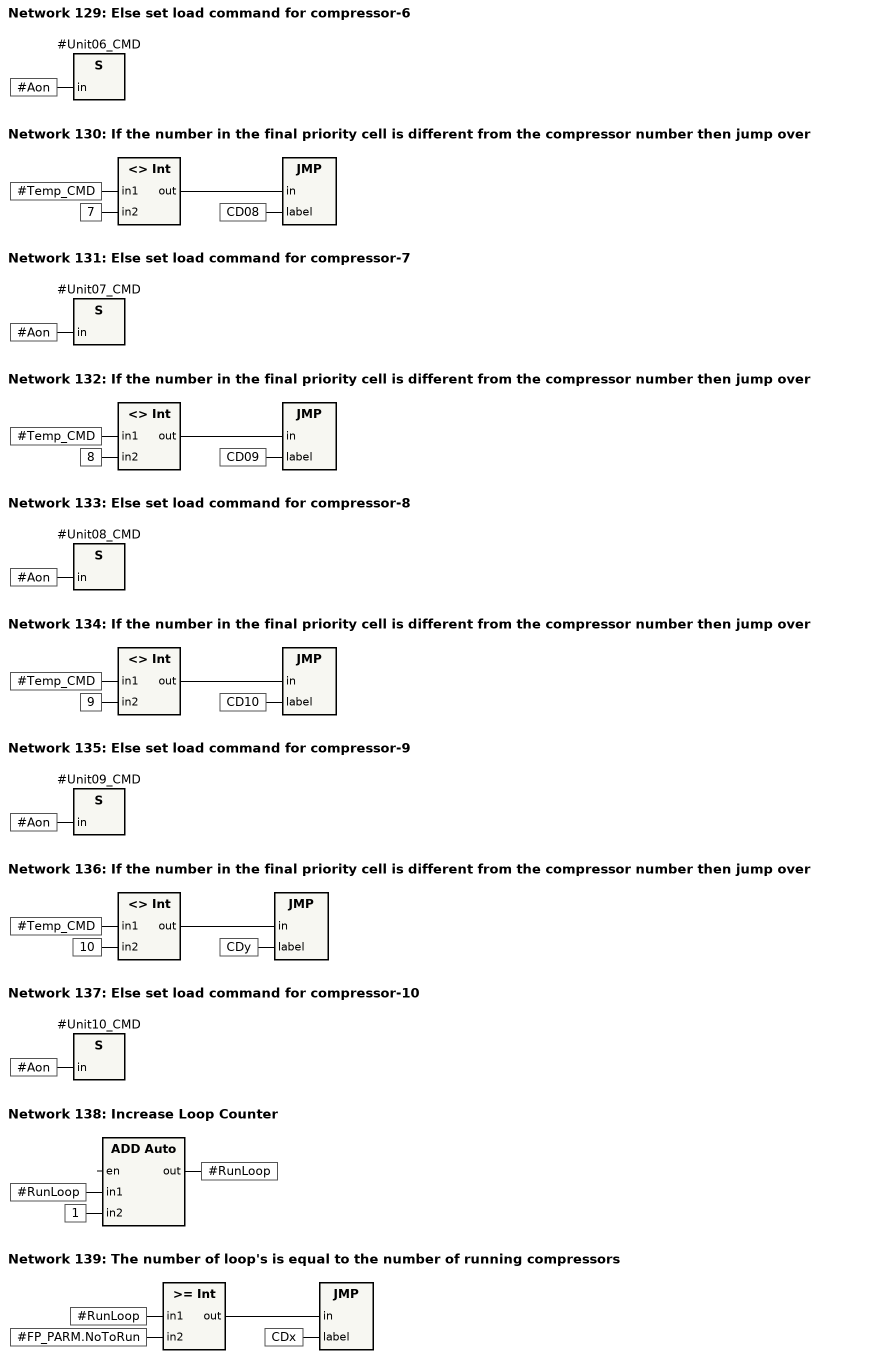
   IF #Aon THEN #Unit06_CMD := TRUE; END_IF;
END_REGION

REGION Network 130: If the number in the final priority cell is different from the compressor number then jump over
   CD07:
   IF #Temp_CMD <> 7 THEN GOTO CD08; END_IF;
END_REGION

REGION Network 131: Else set load command for compressor-7
   IF #Aon THEN #Unit07_CMD := TRUE; END_IF;
END_REGION

REGION Network 132: If the number in the final priority cell is different from the compressor number then jump over
   CD08:
   IF #Temp_CMD <> 8 THEN GOTO CD09; END_IF;
END_REGION

REGION Network 133: Else set load command for compressor-8
   IF #Aon THEN #Unit08_CMD := TRUE; END_IF;
END_REGION

REGION Network 134: If the number in the final priority cell is different from the compressor number then jump over
   CD09:
   IF #Temp_CMD <> 9 THEN GOTO CD10; END_IF;
END_REGION

REGION Network 135: Else set load command for compressor-9
   IF #Aon THEN #Unit09_CMD := TRUE; END_IF;
END_REGION

REGION Network 136: If the number in the final priority cell is different from the compressor number then jump over
   CD10:
   IF #Temp_CMD <> 10 THEN GOTO CDy; END_IF;
END_REGION

REGION Network 137: Else set load command for compressor-10
   IF #Aon THEN #Unit10_CMD := TRUE; END_IF;
END_REGION

REGION Network 138: Increase Loop Counter
   CDy:
   #RunLoop := #RunLoop + 1;
END_REGION

REGION Network 139: The number of loop's is equal to the number of running compressors
   IF #RunLoop >= #FP_PARM.NoToRun THEN GOTO CDx; END_IF;
END_REGION

REGION Network 140: pointer to the next priority cell
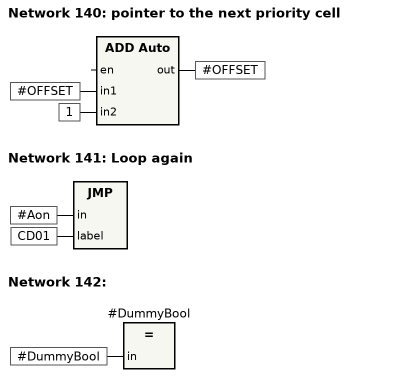
   #OFFSET := #OFFSET + 1;
END_REGION

REGION Network 141: Loop again
   IF #Aon THEN GOTO CD01; END_IF;
END_REGION

REGION Network 142
   CDx:
   #DummyBool := #DummyBool;
END_REGION

REGION Network 143: Check to determine if change is in progress
   // If difference between Comm and Load change is in progress 
   // then set priorityprogress flag
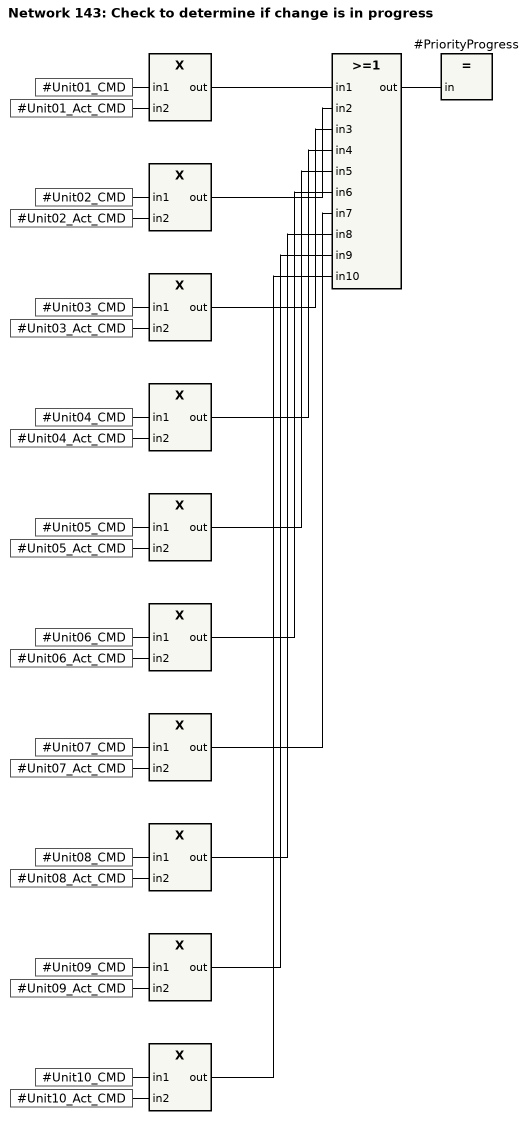
   #PriorityProgress := (#Unit01_CMD XOR #Unit01_Act_CMD) OR (#Unit02_CMD XOR #Unit02_Act_CMD) OR (#Unit03_CMD XOR #Unit03_Act_CMD) OR (#Unit04_CMD XOR #Unit04_Act_CMD) OR (#Unit05_CMD XOR #Unit05_Act_CMD) OR (#Unit06_CMD XOR #Unit06_Act_CMD) OR (#Unit07_CMD XOR #Unit07_Act_CMD) OR (#Unit08_CMD XOR #Unit08_Act_CMD) OR (#Unit09_CMD XOR #Unit09_Act_CMD) OR (#Unit10_CMD XOR #Unit10_Act_CMD);
END_REGION

REGION Network 144: Wait for Run Delay before stopping
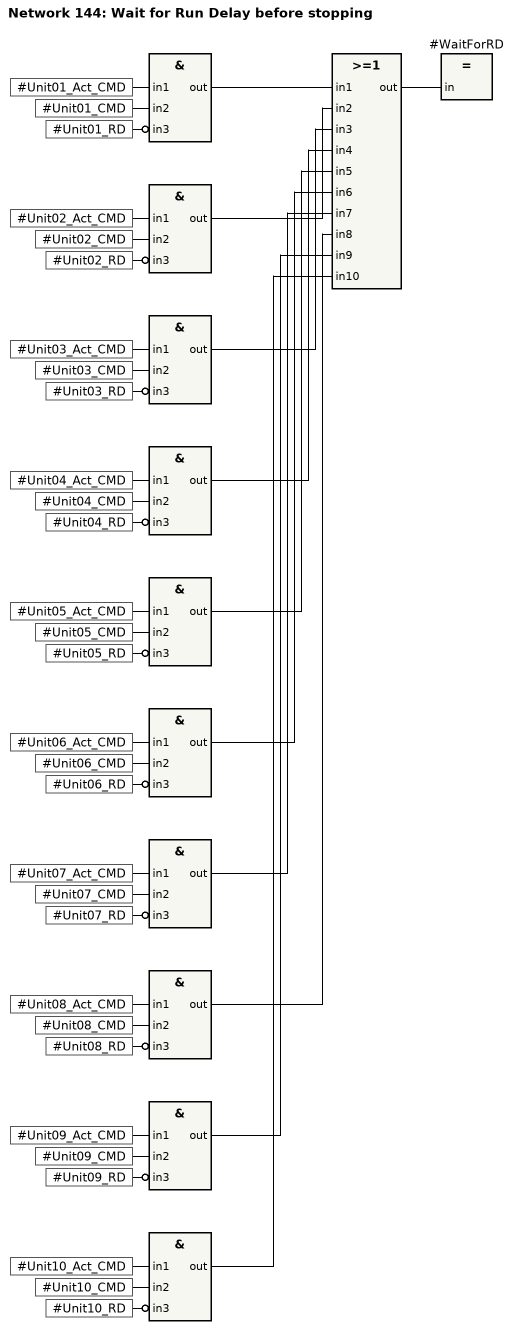
   #WaitForRD := (#Unit01_Act_CMD AND #Unit01_CMD AND NOT #Unit01_RD) OR (#Unit02_Act_CMD AND #Unit02_CMD AND NOT #Unit02_RD) OR (#Unit03_Act_CMD AND #Unit03_CMD AND NOT #Unit03_RD) OR (#Unit04_Act_CMD AND #Unit04_CMD AND NOT #Unit04_RD) OR (#Unit05_Act_CMD AND #Unit05_CMD AND NOT #Unit05_RD) OR (#Unit06_Act_CMD AND #Unit06_CMD AND NOT #Unit06_RD) OR (#Unit07_Act_CMD AND #Unit07_CMD AND NOT #Unit07_RD) OR (#Unit08_Act_CMD AND #Unit08_CMD AND NOT #Unit08_RD) OR (#Unit09_Act_CMD AND #Unit09_CMD AND NOT #Unit09_RD) OR (#Unit10_Act_CMD AND #Unit10_CMD AND NOT #Unit10_RD);
END_REGION

REGION Network 145: Timer to ensure selectivity
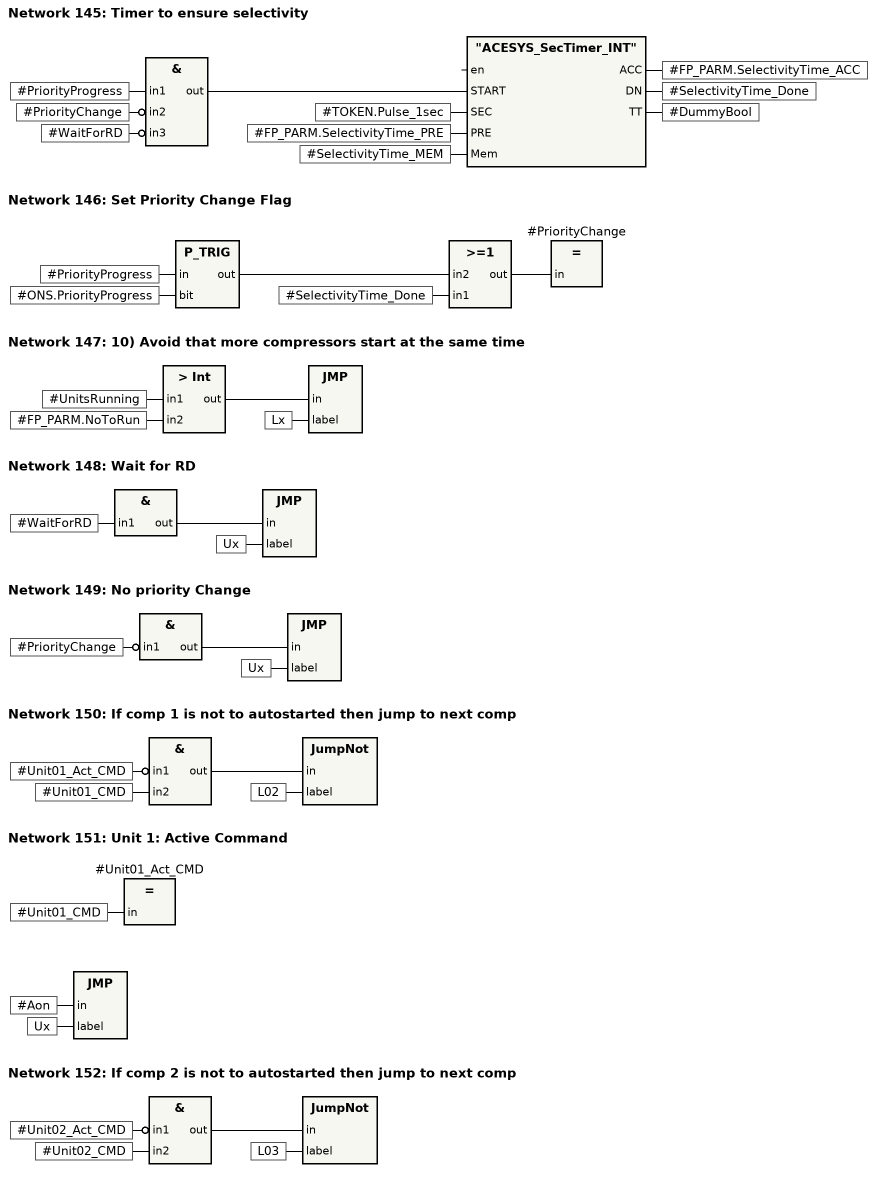
   "ACESYS_SecTimer_INT"(START := #PriorityProgress AND NOT #PriorityChange AND NOT #WaitForRD,
                         SEC := #TOKEN.Pulse_1sec,
                         PRE := #FP_PARM.SelectivityTime_PRE,
                         Mem := #SelectivityTime_MEM,
                         ACC => #FP_PARM.SelectivityTime_ACC,
                         DN => #SelectivityTime_Done,
                         TT => #DummyBool);
END_REGION

REGION Network 146: Set Priority Change Flag
   #_w1 := #PriorityProgress AND NOT #ONS.PriorityProgress;   // rising edge
   #ONS.PriorityProgress := #PriorityProgress;
   #PriorityChange := #_w1 OR #SelectivityTime_Done;
END_REGION

REGION Network 147: 10) Avoid that more compressors start at the same time
   // Every x s a compressor is loaded
   IF #UnitsRunning > #FP_PARM.NoToRun THEN GOTO Lx; END_IF;
END_REGION

REGION Network 148: Wait for RD
   IF #WaitForRD THEN GOTO Ux; END_IF;
END_REGION

REGION Network 149: No priority Change
   IF NOT #PriorityChange THEN GOTO Ux; END_IF;
END_REGION

REGION Network 150: If comp 1 is not to autostarted then jump to next comp
   // no SCL statement known for JumpNot: written as a call
   JumpNot(in := NOT #Unit01_Act_CMD AND #Unit01_CMD, label := L02);
END_REGION

REGION Network 151: Unit 1: Active Command
   // Jump to end
   #Unit01_Act_CMD := #Unit01_CMD;
   IF #Aon THEN GOTO Ux; END_IF;
END_REGION

REGION Network 152: If comp 2 is not to autostarted then jump to next comp
   // no SCL statement known for JumpNot: written as a call
   L02:
   JumpNot(in := NOT #Unit02_Act_CMD AND #Unit02_CMD, label := L03);
END_REGION

REGION Network 153: Unit 2: Active Command
   // Jump to end
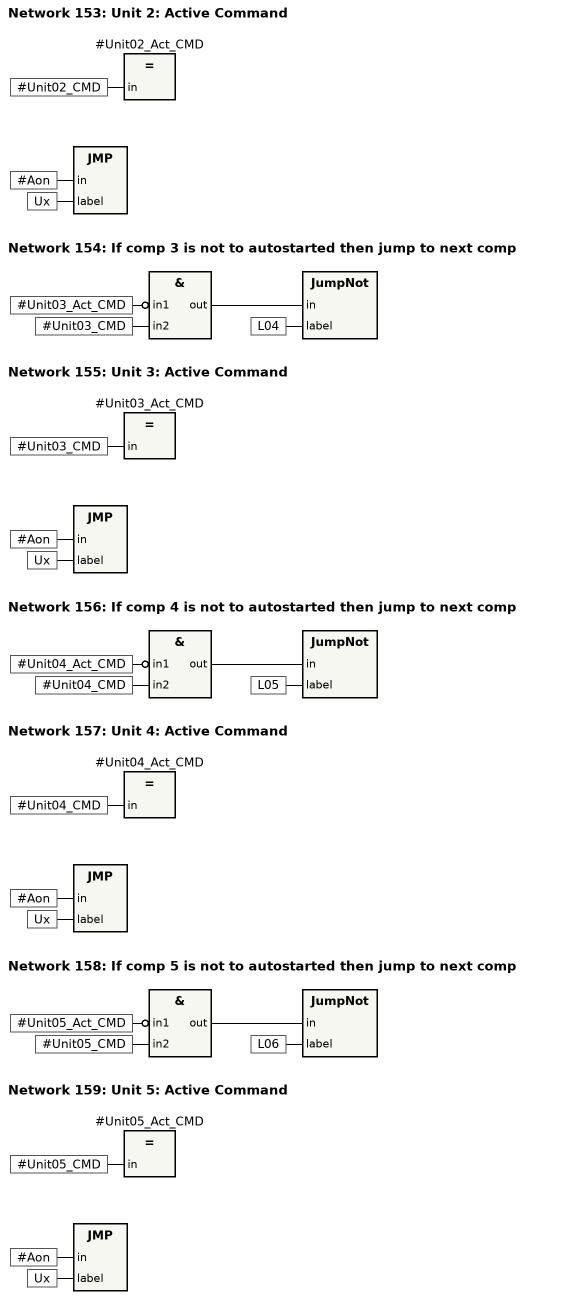
   #Unit02_Act_CMD := #Unit02_CMD;
   IF #Aon THEN GOTO Ux; END_IF;
END_REGION

REGION Network 154: If comp 3 is not to autostarted then jump to next comp
   // no SCL statement known for JumpNot: written as a call
   L03:
   JumpNot(in := NOT #Unit03_Act_CMD AND #Unit03_CMD, label := L04);
END_REGION

REGION Network 155: Unit 3: Active Command
   // Jump to end
   #Unit03_Act_CMD := #Unit03_CMD;
   IF #Aon THEN GOTO Ux; END_IF;
END_REGION

REGION Network 156: If comp 4 is not to autostarted then jump to next comp
   // no SCL statement known for JumpNot: written as a call
   L04:
   JumpNot(in := NOT #Unit04_Act_CMD AND #Unit04_CMD, label := L05);
END_REGION

REGION Network 157: Unit 4: Active Command
   // Jump to end
   #Unit04_Act_CMD := #Unit04_CMD;
   IF #Aon THEN GOTO Ux; END_IF;
END_REGION

REGION Network 158: If comp 5 is not to autostarted then jump to next comp
   // no SCL statement known for JumpNot: written as a call
   L05:
   JumpNot(in := NOT #Unit05_Act_CMD AND #Unit05_CMD, label := L06);
END_REGION

REGION Network 159: Unit 5: Active Command
   // Jump to end
   #Unit05_Act_CMD := #Unit05_CMD;
   IF #Aon THEN GOTO Ux; END_IF;
END_REGION

REGION Network 160: If comp 6 is not to autostarted then jump to next comp
